TYPE "UDT_WSGConfiguration"
VERSION : 0.1
   STRUCT
      GlobalConfig { ExternalAccessible := 'False'; ExternalVisible := 'False'; ExternalWritable := 'False'} : Struct
         LeftStationExists { ExternalAccessible := 'False'; ExternalVisible := 'False'; ExternalWritable := 'False'} : Bool := TRUE;
         RightStationExists { ExternalAccessible := 'False'; ExternalVisible := 'False'; ExternalWritable := 'False'} : Bool := TRUE;
      END_STRUCT;
      "010" { ExternalAccessible := 'False'; ExternalVisible := 'False'; ExternalWritable := 'False'} : Struct
         Conveyor { ExternalAccessible := 'False'; ExternalVisible := 'False'; ExternalWritable := 'False'; S7_SetPoint := 'False'} : "UDT_ConveyorConfiguration" := (((), ()), (), (), 100, (), 500, 1000, FALSE, ());
         PEC_Eos { ExternalAccessible := 'False'; ExternalVisible := 'False'; ExternalWritable := 'False'; S7_SetPoint := 'False'} : "UDT_PECConfiguration";
         MCO_M01 { ExternalAccessible := 'False'; ExternalVisible := 'False'; ExternalWritable := 'False'; S7_SetPoint := 'False'} : "UDT_AixPlcFullControllerConfiguration";
      END_STRUCT;
      "020" { ExternalAccessible := 'False'; ExternalVisible := 'False'; ExternalWritable := 'False'} : Struct
         Conveyor { ExternalAccessible := 'False'; ExternalVisible := 'False'; ExternalWritable := 'False'; S7_SetPoint := 'False'} : "UDT_ConveyorConfiguration" := (((), ()), (), (), 100, 0, 500, 1000, FALSE, FALSE);
         PEC_EoS { ExternalAccessible := 'False'; ExternalVisible := 'False'; ExternalWritable := 'False'} : "UDT_PECConfiguration";
         MCO_M01 { ExternalAccessible := 'False'; ExternalVisible := 'False'; ExternalWritable := 'False'; S7_SetPoint := 'False'} : "UDT_AixPlcFullControllerConfiguration";
      END_STRUCT;
      "021" { ExternalAccessible := 'False'; ExternalVisible := 'False'; ExternalWritable := 'False'} : Struct
         Conveyor { ExternalAccessible := 'False'; ExternalVisible := 'False'; ExternalWritable := 'False'; S7_SetPoint := 'False'} : "UDT_ConveyorConfiguration" := (((), ()), (), (), 100, 0, 500, 1000, FALSE, FALSE);
         RightAngledTransfer { ExternalAccessible := 'False'; ExternalVisible := 'False'; ExternalWritable := 'False'; S7_SetPoint := 'False'} : "UDT_RATConfiguration";
         MCO_M01 { ExternalAccessible := 'False'; ExternalVisible := 'False'; ExternalWritable := 'False'; S7_SetPoint := 'False'} : "UDT_AixPlcFullControllerConfiguration";
      END_STRUCT;
      "110" { ExternalAccessible := 'False'; ExternalVisible := 'False'; ExternalWritable := 'False'} : Struct
         Conveyor { ExternalAccessible := 'False'; ExternalVisible := 'False'; ExternalWritable := 'False'; S7_SetPoint := 'False'} : "UDT_ConveyorConfiguration" := (((), ()), (), (), (), (), 500, 1000, FALSE, ());
         PEC_Eos { ExternalAccessible := 'False'; ExternalVisible := 'False'; ExternalWritable := 'False'} : "UDT_PECUpdateConfiguration";
         MCO_M01 { ExternalAccessible := 'False'; ExternalVisible := 'False'; ExternalWritable := 'False'} : "UDT_AixPlcFullControllerConfiguration";
      END_STRUCT;
      "120" { ExternalAccessible := 'False'; ExternalVisible := 'False'; ExternalWritable := 'False'} : Struct
         Conveyor { ExternalAccessible := 'False'; ExternalVisible := 'False'; ExternalWritable := 'False'; S7_SetPoint := 'False'} : "UDT_ConveyorConfiguration" := (((), ()), (), (), (), (), 500, 1000, FALSE, ());
         MCO_M01 { ExternalAccessible := 'False'; ExternalVisible := 'False'; ExternalWritable := 'False'} : "UDT_AixPlcFullControllerConfiguration";
      END_STRUCT;
      "130" { ExternalAccessible := 'False'; ExternalVisible := 'False'; ExternalWritable := 'False'} : Struct
         Conveyor { ExternalAccessible := 'False'; ExternalVisible := 'False'; ExternalWritable := 'False'; S7_SetPoint := 'False'} : "UDT_ConveyorConfiguration" := (((), ()), (), (), 100, (), 500, 1000, FALSE, ());
         PEC_Eos { ExternalAccessible := 'False'; ExternalVisible := 'False'; ExternalWritable := 'False'} : "UDT_PECUpdateConfiguration";
         MCO_M01 { ExternalAccessible := 'False'; ExternalVisible := 'False'; ExternalWritable := 'False'} : "UDT_AixPlcFullControllerConfiguration";
      END_STRUCT;
      "140" { ExternalAccessible := 'False'; ExternalVisible := 'False'; ExternalWritable := 'False'} : Struct
         Conveyor { ExternalAccessible := 'False'; ExternalVisible := 'False'; ExternalWritable := 'False'} : "UDT_ConveyorConfiguration" := (((), ()), (), (), 100, 0, 500, 1000, FALSE, FALSE);
         PEC_EoS { ExternalAccessible := 'False'; ExternalVisible := 'False'; ExternalWritable := 'False'} : "UDT_PECConfiguration";
         MCO_M01 { ExternalAccessible := 'False'; ExternalVisible := 'False'; ExternalWritable := 'False'} : "UDT_AixPlcFullControllerConfiguration";
      END_STRUCT;
      "141" { ExternalAccessible := 'False'; ExternalVisible := 'False'; ExternalWritable := 'False'} : Struct
         Conveyor { ExternalAccessible := 'False'; ExternalVisible := 'False'; ExternalWritable := 'False'; S7_SetPoint := 'False'} : "UDT_ConveyorConfiguration" := (((), ()), (), (), 100, 0, 500, 1000, FALSE, FALSE);
         RightAngledTransfer { ExternalAccessible := 'False'; ExternalVisible := 'False'; ExternalWritable := 'False'} : "UDT_RATConfiguration";
         MCO_M01 { ExternalAccessible := 'False'; ExternalVisible := 'False'; ExternalWritable := 'False'} : "UDT_AixPlcFullControllerConfiguration";
      END_STRUCT;
      "150" { ExternalAccessible := 'False'; ExternalVisible := 'False'; ExternalWritable := 'False'} : Struct
         Conveyor { ExternalAccessible := 'False'; ExternalVisible := 'False'; ExternalWritable := 'False'; S7_SetPoint := 'False'} : "UDT_ConveyorConfiguration" := (((), ()), (), (), 100, (), 500, 1000, FALSE, ());
         PEC_Eos { ExternalAccessible := 'False'; ExternalVisible := 'False'; ExternalWritable := 'False'} : "UDT_PECUpdateConfiguration" := (600, 300, 5, 5, (), (), 50, 50, (), (), (), 1, 5, (), (), (), ());
         MCO_M01 { ExternalAccessible := 'False'; ExternalVisible := 'False'; ExternalWritable := 'False'} : "UDT_AixPlcFullControllerConfiguration";
      END_STRUCT;
      "160" { ExternalAccessible := 'False'; ExternalVisible := 'False'; ExternalWritable := 'False'} : Struct
         Conveyor { ExternalAccessible := 'False'; ExternalVisible := 'False'; ExternalWritable := 'False'; S7_SetPoint := 'False'} : "UDT_ConveyorConfiguration" := (((), ()), (), (), 100, 0, 500, 1000, FALSE, FALSE);
         PEC_Eos { ExternalAccessible := 'False'; ExternalVisible := 'False'; ExternalWritable := 'False'} : "UDT_PECUpdateConfiguration" := (600, 300, 5, 5, TRUE, FALSE, 50, 50, 1, 5, 0, 1, 5, FALSE, FALSE, FALSE, FALSE);
         MCO_M01 { ExternalAccessible := 'False'; ExternalVisible := 'False'; ExternalWritable := 'False'} : "UDT_AixPlcFullControllerConfiguration";
      END_STRUCT;
      "170" { ExternalAccessible := 'False'; ExternalVisible := 'False'; ExternalWritable := 'False'} : Struct
         Conveyor { ExternalAccessible := 'False'; ExternalVisible := 'False'; ExternalWritable := 'False'; S7_SetPoint := 'False'} : "UDT_ConveyorConfiguration" := (((), ()), (), (), 100, (), 500, 1000, FALSE, ());
         PEC_Eos { ExternalAccessible := 'False'; ExternalVisible := 'False'; ExternalWritable := 'False'} : "UDT_PECUpdateConfiguration" := (600, 300, 5, 5, (), (), 50, 50, (), (), (), 1, 5, (), (), (), ());
         MCO_M01 { ExternalAccessible := 'False'; ExternalVisible := 'False'; ExternalWritable := 'False'} : "UDT_AixPlcFullControllerConfiguration";
      END_STRUCT;
      "180" { ExternalAccessible := 'False'; ExternalVisible := 'False'; ExternalWritable := 'False'} : Struct
         Conveyor { ExternalAccessible := 'False'; ExternalVisible := 'False'; ExternalWritable := 'False'; S7_SetPoint := 'False'} : "UDT_ConveyorConfiguration" := (((), ()), (), (), 100, (), 500, 1000, FALSE, ());
         PEC_Eos { ExternalAccessible := 'False'; ExternalVisible := 'False'; ExternalWritable := 'False'} : "UDT_PECUpdateConfiguration" := (600, 300, 5, 5, (), (), 50, 50, (), (), (), 1, 5, (), (), (), ());
         MCO_M01 { ExternalAccessible := 'False'; ExternalVisible := 'False'; ExternalWritable := 'False'} : "UDT_AixPlcFullControllerConfiguration";
      END_STRUCT;
      "190" { ExternalAccessible := 'False'; ExternalVisible := 'False'; ExternalWritable := 'False'} : Struct
         Conveyor { ExternalAccessible := 'False'; ExternalVisible := 'False'; ExternalWritable := 'False'; S7_SetPoint := 'False'} : "UDT_ConveyorConfiguration" := (((), ()), (), (), 100, (), 500, 1000, FALSE, ());
         PEC_Eos { ExternalAccessible := 'False'; ExternalVisible := 'False'; ExternalWritable := 'False'} : "UDT_PECUpdateConfiguration" := (600, 300, 5, 5, (), (), 50, 50, (), (), (), 1, 5, (), (), (), ());
         MCO_M01 { ExternalAccessible := 'False'; ExternalVisible := 'False'; ExternalWritable := 'False'} : "UDT_AixPlcFullControllerConfiguration";
      END_STRUCT;
      "210" { ExternalAccessible := 'False'; ExternalVisible := 'False'; ExternalWritable := 'False'} : Struct
         Conveyor { ExternalAccessible := 'False'; ExternalVisible := 'False'; ExternalWritable := 'False'; S7_SetPoint := 'False'} : "UDT_ConveyorConfiguration" := (((), ()), (), (), 100, 0, 500, 1000, FALSE, FALSE);
         PEC_EoS { ExternalAccessible := 'False'; ExternalVisible := 'False'; ExternalWritable := 'False'} : "UDT_PECConfiguration";
         MCO_M01 { ExternalAccessible := 'False'; ExternalVisible := 'False'; ExternalWritable := 'False'} : "UDT_AixPlcFullControllerConfiguration";
      END_STRUCT;
      "211" { ExternalAccessible := 'False'; ExternalVisible := 'False'; ExternalWritable := 'False'} : Struct
         Conveyor { ExternalAccessible := 'False'; ExternalVisible := 'False'; ExternalWritable := 'False'; S7_SetPoint := 'False'} : "UDT_ConveyorConfiguration" := (((), ()), (), (), 100, 0, 500, 1000, FALSE, FALSE);
         RightAngledTransfer { ExternalAccessible := 'False'; ExternalVisible := 'False'; ExternalWritable := 'False'} : "UDT_RATConfiguration";
         MCO_M01 { ExternalAccessible := 'False'; ExternalVisible := 'False'; ExternalWritable := 'False'} : "UDT_AixPlcFullControllerConfiguration";
      END_STRUCT;
      "220" { ExternalAccessible := 'False'; ExternalVisible := 'False'; ExternalWritable := 'False'} : Struct
         Conveyor { ExternalAccessible := 'False'; ExternalVisible := 'False'; ExternalWritable := 'False'} : "UDT_ConveyorConfiguration" := (((), ()), (), (), 100, 0, 500, 1000, FALSE, FALSE);
         PEC_EoS { ExternalAccessible := 'False'; ExternalVisible := 'False'; ExternalWritable := 'False'} : "UDT_PECConfiguration";
         MCO_M01 { ExternalAccessible := 'False'; ExternalVisible := 'False'; ExternalWritable := 'False'} : "UDT_AixPlcFullControllerConfiguration";
      END_STRUCT;
      "221" { ExternalAccessible := 'False'; ExternalVisible := 'False'; ExternalWritable := 'False'} : Struct
         Conveyor { ExternalAccessible := 'False'; ExternalVisible := 'False'; ExternalWritable := 'False'; S7_SetPoint := 'False'} : "UDT_ConveyorConfiguration" := (((), ()), (), (), 100, 0, 500, 1000, FALSE, FALSE);
         RightAngledTransfer { ExternalAccessible := 'False'; ExternalVisible := 'False'; ExternalWritable := 'False'} : "UDT_RATConfiguration";
         MCO_M01 { ExternalAccessible := 'False'; ExternalVisible := 'False'; ExternalWritable := 'False'} : "UDT_AixPlcFullControllerConfiguration";
      END_STRUCT;
      "230" { ExternalAccessible := 'False'; ExternalVisible := 'False'; ExternalWritable := 'False'} : Struct
         Conveyor { ExternalAccessible := 'False'; ExternalVisible := 'False'; ExternalWritable := 'False'; S7_SetPoint := 'False'} : "UDT_ConveyorConfiguration" := (((), ()), (), (), 100, (), 500, 1000, FALSE, ());
         MCO_M01 { ExternalAccessible := 'False'; ExternalVisible := 'False'; ExternalWritable := 'False'} : "UDT_AixPlcFullControllerConfiguration";
      END_STRUCT;
      "310" { ExternalAccessible := 'False'; ExternalVisible := 'False'; ExternalWritable := 'False'} : Struct
         Conveyor { ExternalAccessible := 'False'; ExternalVisible := 'False'; ExternalWritable := 'False'; S7_SetPoint := 'False'} : "UDT_ConveyorConfiguration" := (((), ()), (), (), 100, (), 500, 1000, FALSE, ());
         PEC_Eos { ExternalAccessible := 'False'; ExternalVisible := 'False'; ExternalWritable := 'False'} : "UDT_PECConfiguration" := (600, 300, 5, 5, ());
         MCO_M01 { ExternalAccessible := 'False'; ExternalVisible := 'False'; ExternalWritable := 'False'} : "UDT_AixPlcFullControllerConfiguration";
      END_STRUCT;
      "320" { ExternalAccessible := 'False'; ExternalVisible := 'False'; ExternalWritable := 'False'} : Struct
         Conveyor { ExternalAccessible := 'False'; ExternalVisible := 'False'; ExternalWritable := 'False'; S7_SetPoint := 'False'} : "UDT_ConveyorConfiguration" := (((), ()), (), (), 100, (), 500, 1000, FALSE, ());
         PEC_Eos { ExternalAccessible := 'False'; ExternalVisible := 'False'; ExternalWritable := 'False'} : "UDT_PECConfiguration" := (600, 300, 5, 5, ());
         MCO_M01 { ExternalAccessible := 'False'; ExternalVisible := 'False'; ExternalWritable := 'False'} : "UDT_AixPlcFullControllerConfiguration";
      END_STRUCT;
      "330" { ExternalAccessible := 'False'; ExternalVisible := 'False'; ExternalWritable := 'False'} : Struct
         Conveyor { ExternalAccessible := 'False'; ExternalVisible := 'False'; ExternalWritable := 'False'; S7_SetPoint := 'False'} : "UDT_ConveyorConfiguration" := (((), ()), (), (), 100, (), 500, 1000, FALSE, ());
         PEC_Eos { ExternalAccessible := 'False'; ExternalVisible := 'False'; ExternalWritable := 'False'} : "UDT_PECConfiguration" := (600, 300, 5, 5, ());
         MCO_M01 { ExternalAccessible := 'False'; ExternalVisible := 'False'; ExternalWritable := 'False'} : "UDT_AixPlcFullControllerConfiguration";
      END_STRUCT;
      "340" { ExternalAccessible := 'False'; ExternalVisible := 'False'; ExternalWritable := 'False'} : Struct
         Conveyor { ExternalAccessible := 'False'; ExternalVisible := 'False'; ExternalWritable := 'False'; S7_SetPoint := 'False'} : "UDT_ConveyorConfiguration" := (((), ()), (), (), 100, (), 500, 1000, FALSE, ());
         PEC_Eos { ExternalAccessible := 'False'; ExternalVisible := 'False'; ExternalWritable := 'False'} : "UDT_PECConfiguration" := (600, 300, 5, 5, ());
         MCO_M01 { ExternalAccessible := 'False'; ExternalVisible := 'False'; ExternalWritable := 'False'} : "UDT_AixPlcFullControllerConfiguration";
      END_STRUCT;
      "350" { ExternalAccessible := 'False'; ExternalVisible := 'False'; ExternalWritable := 'False'} : Struct
         Conveyor { ExternalAccessible := 'False'; ExternalVisible := 'False'; ExternalWritable := 'False'; S7_SetPoint := 'False'} : "UDT_ConveyorConfiguration" := (((), ()), (), (), 100, (), 500, 1000, FALSE, ());
         PEC_Eos { ExternalAccessible := 'False'; ExternalVisible := 'False'; ExternalWritable := 'False'} : "UDT_PECConfiguration" := (600, 300, 5, 5, ());
         MCO_M01 { ExternalAccessible := 'False'; ExternalVisible := 'False'; ExternalWritable := 'False'} : "UDT_AixPlcFullControllerConfiguration";
      END_STRUCT;
      "510" { ExternalAccessible := 'False'; ExternalVisible := 'False'; ExternalWritable := 'False'} : Struct
         Conveyor { ExternalAccessible := 'False'; ExternalVisible := 'False'; ExternalWritable := 'False'; S7_SetPoint := 'False'} : "UDT_ConveyorConfiguration" := (((), ()), (), (), 100, (), 500, 1000, FALSE, ());
         MCO_M01 { ExternalAccessible := 'False'; ExternalVisible := 'False'; ExternalWritable := 'False'} : "UDT_AixPlcFullControllerConfiguration";
      END_STRUCT;
      "520" { ExternalAccessible := 'False'; ExternalVisible := 'False'; ExternalWritable := 'False'} : Struct
         Conveyor { ExternalAccessible := 'False'; ExternalVisible := 'False'; ExternalWritable := 'False'; S7_SetPoint := 'False'} : "UDT_ConveyorConfiguration" := (((), ()), (), (), 100, (), 500, 1000, FALSE, ());
         PEC_Eos { ExternalAccessible := 'False'; ExternalVisible := 'False'; ExternalWritable := 'False'; S7_SetPoint := 'False'} : "UDT_PECUpdateConfiguration";
         MCO_M01 { ExternalAccessible := 'False'; ExternalVisible := 'False'; ExternalWritable := 'False'} : "UDT_AixPlcFullControllerConfiguration";
      END_STRUCT;
      "530" { ExternalAccessible := 'False'; ExternalVisible := 'False'; ExternalWritable := 'False'} : Struct
         Conveyor { ExternalAccessible := 'False'; ExternalVisible := 'False'; ExternalWritable := 'False'; S7_SetPoint := 'False'} : "UDT_ConveyorConfiguration" := (((), ()), (), (), 100, (), 500, 1000, FALSE, ());
         PEC_Eos { ExternalAccessible := 'False'; ExternalVisible := 'False'; ExternalWritable := 'False'; S7_SetPoint := 'False'} : "UDT_PECUpdateConfiguration";
         MCO_M01 { ExternalAccessible := 'False'; ExternalVisible := 'False'; ExternalWritable := 'False'} : "UDT_AixPlcFullControllerConfiguration";
      END_STRUCT;
      "540" { ExternalAccessible := 'False'; ExternalVisible := 'False'; ExternalWritable := 'False'} : Struct
         Conveyor { ExternalAccessible := 'False'; ExternalVisible := 'False'; ExternalWritable := 'False'} : "UDT_ConveyorConfiguration" := (((), ()), (), (), 100, 0, 500, 1000, FALSE, FALSE);
         PEC_EoS { ExternalAccessible := 'False'; ExternalVisible := 'False'; ExternalWritable := 'False'} : "UDT_PECConfiguration";
         MCO_M01 { ExternalAccessible := 'False'; ExternalVisible := 'False'; ExternalWritable := 'False'} : "UDT_AixPlcFullControllerConfiguration";
      END_STRUCT;
      "541" { ExternalAccessible := 'False'; ExternalVisible := 'False'; ExternalWritable := 'False'} : Struct
         Conveyor { ExternalAccessible := 'False'; ExternalVisible := 'False'; ExternalWritable := 'False'} : "UDT_ConveyorConfiguration" := (((), ()), (), (), 100, 0, 500, 1000, FALSE, FALSE);
         RightAngledTransfer { ExternalAccessible := 'False'; ExternalVisible := 'False'; ExternalWritable := 'False'} : "UDT_RATConfiguration";
         MCO_M01 { ExternalAccessible := 'False'; ExternalVisible := 'False'; ExternalWritable := 'False'} : "UDT_AixPlcFullControllerConfiguration";
      END_STRUCT;
      "550" { ExternalAccessible := 'False'; ExternalVisible := 'False'; ExternalWritable := 'False'} : Struct
         Conveyor { ExternalAccessible := 'False'; ExternalVisible := 'False'; ExternalWritable := 'False'; S7_SetPoint := 'False'} : "UDT_ConveyorConfiguration" := (((), ()), (), (), 100, (), 500, 1000, FALSE, ());
         PEC_Eos { ExternalAccessible := 'False'; ExternalVisible := 'False'; ExternalWritable := 'False'} : "UDT_PECUpdateConfiguration" := (600, 300, 5, 5, (), (), 50, 50, (), (), (), 1, 5, (), (), (), ());
         MCO_M01 { ExternalAccessible := 'False'; ExternalVisible := 'False'; ExternalWritable := 'False'} : "UDT_AixPlcFullControllerConfiguration";
      END_STRUCT;
      "560" { ExternalAccessible := 'False'; ExternalVisible := 'False'; ExternalWritable := 'False'} : Struct
         Conveyor { ExternalAccessible := 'False'; ExternalVisible := 'False'; ExternalWritable := 'False'; S7_SetPoint := 'False'} : "UDT_ConveyorConfiguration" := (((), ()), (), (), 100, 0, 500, 1000, FALSE, FALSE);
         PEC_Eos { ExternalAccessible := 'False'; ExternalVisible := 'False'; ExternalWritable := 'False'} : "UDT_PECUpdateConfiguration" := (600, 300, 5, 5, TRUE, FALSE, 50, 50, 1, 5, 0, 1, 5, FALSE, FALSE, FALSE, FALSE);
         MCO_M01 { ExternalAccessible := 'False'; ExternalVisible := 'False'; ExternalWritable := 'False'} : "UDT_AixPlcFullControllerConfiguration";
      END_STRUCT;
      "570" { ExternalAccessible := 'False'; ExternalVisible := 'False'; ExternalWritable := 'False'} : Struct
         Conveyor { ExternalAccessible := 'False'; ExternalVisible := 'False'; ExternalWritable := 'False'; S7_SetPoint := 'False'} : "UDT_ConveyorConfiguration" := (((), ()), (), (), 100, (), 500, 1000, FALSE, ());
         PEC_Eos { ExternalAccessible := 'False'; ExternalVisible := 'False'; ExternalWritable := 'False'} : "UDT_PECUpdateConfiguration" := (600, 300, 5, 5, (), (), 50, 50, (), (), (), 1, 5, (), (), (), ());
         MCO_M01 { ExternalAccessible := 'False'; ExternalVisible := 'False'; ExternalWritable := 'False'} : "UDT_AixPlcFullControllerConfiguration";
      END_STRUCT;
      "580" { ExternalAccessible := 'False'; ExternalVisible := 'False'; ExternalWritable := 'False'} : Struct
         Conveyor { ExternalAccessible := 'False'; ExternalVisible := 'False'; ExternalWritable := 'False'; S7_SetPoint := 'False'} : "UDT_ConveyorConfiguration" := (((), ()), (), (), 100, (), 500, 1000, FALSE, ());
         PEC_Eos { ExternalAccessible := 'False'; ExternalVisible := 'False'; ExternalWritable := 'False'} : "UDT_PECUpdateConfiguration" := (600, 300, 5, 5, (), (), 50, 50, (), (), (), 1, 5, (), (), (), ());
         MCO_M01 { ExternalAccessible := 'False'; ExternalVisible := 'False'; ExternalWritable := 'False'} : "UDT_AixPlcFullControllerConfiguration";
      END_STRUCT;
      "590" { ExternalAccessible := 'False'; ExternalVisible := 'False'; ExternalWritable := 'False'} : Struct
         Conveyor { ExternalAccessible := 'False'; ExternalVisible := 'False'; ExternalWritable := 'False'; S7_SetPoint := 'False'} : "UDT_ConveyorConfiguration" := (((), ()), (), (), 100, (), 500, 1000, FALSE, ());
         PEC_Eos { ExternalAccessible := 'False'; ExternalVisible := 'False'; ExternalWritable := 'False'} : "UDT_PECUpdateConfiguration" := (600, 300, 5, 5, (), (), 50, 50, (), (), (), 1, 5, (), (), (), ());
         MCO_M01 { ExternalAccessible := 'False'; ExternalVisible := 'False'; ExternalWritable := 'False'} : "UDT_AixPlcFullControllerConfiguration";
      END_STRUCT;
      "610" { ExternalAccessible := 'False'; ExternalVisible := 'False'; ExternalWritable := 'False'} : Struct
         Conveyor { ExternalAccessible := 'False'; ExternalVisible := 'False'; ExternalWritable := 'False'; S7_SetPoint := 'False'} : "UDT_ConveyorConfiguration" := (((), ()), (), (), 100, 0, 500, 1000, FALSE, FALSE);
         PEC_EoS { ExternalAccessible := 'False'; ExternalVisible := 'False'; ExternalWritable := 'False'} : "UDT_PECConfiguration";
         MCO_M01 { ExternalAccessible := 'False'; ExternalVisible := 'False'; ExternalWritable := 'False'} : "UDT_AixPlcFullControllerConfiguration";
      END_STRUCT;
      "611" { ExternalAccessible := 'False'; ExternalVisible := 'False'; ExternalWritable := 'False'} : Struct
         Conveyor { ExternalAccessible := 'False'; ExternalVisible := 'False'; ExternalWritable := 'False'; S7_SetPoint := 'False'} : "UDT_ConveyorConfiguration" := (((), ()), (), (), 100, 0, 500, 1000, FALSE, FALSE);
         RightAngledTransfer { ExternalAccessible := 'False'; ExternalVisible := 'False'; ExternalWritable := 'False'} : "UDT_RATConfiguration";
         MCO_M01 { ExternalAccessible := 'False'; ExternalVisible := 'False'; ExternalWritable := 'False'} : "UDT_AixPlcFullControllerConfiguration";
      END_STRUCT;
      "620" { ExternalAccessible := 'False'; ExternalVisible := 'False'; ExternalWritable := 'False'} : Struct
         Conveyor { ExternalAccessible := 'False'; ExternalVisible := 'False'; ExternalWritable := 'False'} : "UDT_ConveyorConfiguration" := (((), ()), (), (), 100, 0, 500, 1000, FALSE, FALSE);
         PEC_EoS { ExternalAccessible := 'False'; ExternalVisible := 'False'; ExternalWritable := 'False'} : "UDT_PECConfiguration";
         MCO_M01 { ExternalAccessible := 'False'; ExternalVisible := 'False'; ExternalWritable := 'False'} : "UDT_AixPlcFullControllerConfiguration";
      END_STRUCT;
      "621" { ExternalAccessible := 'False'; ExternalVisible := 'False'; ExternalWritable := 'False'} : Struct
         Conveyor { ExternalAccessible := 'False'; ExternalVisible := 'False'; ExternalWritable := 'False'; S7_SetPoint := 'False'} : "UDT_ConveyorConfiguration" := (((), ()), (), (), 100, 0, 500, 1000, FALSE, FALSE);
         RightAngledTransfer { ExternalAccessible := 'False'; ExternalVisible := 'False'; ExternalWritable := 'False'} : "UDT_RATConfiguration";
         MCO_M01 { ExternalAccessible := 'False'; ExternalVisible := 'False'; ExternalWritable := 'False'} : "UDT_AixPlcFullControllerConfiguration";
      END_STRUCT;
      "630" { ExternalAccessible := 'False'; ExternalVisible := 'False'; ExternalWritable := 'False'} : Struct
         Conveyor { ExternalAccessible := 'False'; ExternalVisible := 'False'; ExternalWritable := 'False'; S7_SetPoint := 'False'} : "UDT_ConveyorConfiguration" := (((), ()), (), (), 100, (), 500, 1000, FALSE, ());
         MCO_M01 { ExternalAccessible := 'False'; ExternalVisible := 'False'; ExternalWritable := 'False'} : "UDT_AixPlcFullControllerConfiguration";
      END_STRUCT;
      "710" { ExternalAccessible := 'False'; ExternalVisible := 'False'; ExternalWritable := 'False'} : Struct
         Conveyor { ExternalAccessible := 'False'; ExternalVisible := 'False'; ExternalWritable := 'False'; S7_SetPoint := 'False'} : "UDT_ConveyorConfiguration" := (((), ()), (), (), 100, (), 500, 1000, FALSE, ());
         PEC_Eos { ExternalAccessible := 'False'; ExternalVisible := 'False'; ExternalWritable := 'False'} : "UDT_PECConfiguration" := (600, 300, 5, 5, ());
         MCO_M01 { ExternalAccessible := 'False'; ExternalVisible := 'False'; ExternalWritable := 'False'} : "UDT_AixPlcFullControllerConfiguration";
      END_STRUCT;
      "720" { ExternalAccessible := 'False'; ExternalVisible := 'False'; ExternalWritable := 'False'} : Struct
         Conveyor { ExternalAccessible := 'False'; ExternalVisible := 'False'; ExternalWritable := 'False'; S7_SetPoint := 'False'} : "UDT_ConveyorConfiguration" := (((), ()), (), (), 100, (), 500, 1000, FALSE, ());
         PEC_Eos { ExternalAccessible := 'False'; ExternalVisible := 'False'; ExternalWritable := 'False'} : "UDT_PECConfiguration" := (600, 300, 5, 5, ());
         MCO_M01 { ExternalAccessible := 'False'; ExternalVisible := 'False'; ExternalWritable := 'False'} : "UDT_AixPlcFullControllerConfiguration";
      END_STRUCT;
      "730" { ExternalAccessible := 'False'; ExternalVisible := 'False'; ExternalWritable := 'False'} : Struct
         Conveyor { ExternalAccessible := 'False'; ExternalVisible := 'False'; ExternalWritable := 'False'; S7_SetPoint := 'False'} : "UDT_ConveyorConfiguration" := (((), ()), (), (), 100, (), 500, 1000, FALSE, ());
         PEC_Eos { ExternalAccessible := 'False'; ExternalVisible := 'False'; ExternalWritable := 'False'} : "UDT_PECConfiguration" := (600, 300, 5, 5, ());
         MCO_M01 { ExternalAccessible := 'False'; ExternalVisible := 'False'; ExternalWritable := 'False'} : "UDT_AixPlcFullControllerConfiguration";
      END_STRUCT;
      "740" { ExternalAccessible := 'False'; ExternalVisible := 'False'; ExternalWritable := 'False'} : Struct
         Conveyor { ExternalAccessible := 'False'; ExternalVisible := 'False'; ExternalWritable := 'False'; S7_SetPoint := 'False'} : "UDT_ConveyorConfiguration" := (((), ()), (), (), 100, (), 500, 1000, FALSE, ());
         PEC_Eos { ExternalAccessible := 'False'; ExternalVisible := 'False'; ExternalWritable := 'False'} : "UDT_PECConfiguration" := (600, 300, 5, 5, ());
         MCO_M01 { ExternalAccessible := 'False'; ExternalVisible := 'False'; ExternalWritable := 'False'} : "UDT_AixPlcFullControllerConfiguration";
      END_STRUCT;
      "750" { ExternalAccessible := 'False'; ExternalVisible := 'False'; ExternalWritable := 'False'} : Struct
         Conveyor { ExternalAccessible := 'False'; ExternalVisible := 'False'; ExternalWritable := 'False'; S7_SetPoint := 'False'} : "UDT_ConveyorConfiguration" := (((), ()), (), (), 100, (), 500, 1000, FALSE, ());
         PEC_Eos { ExternalAccessible := 'False'; ExternalVisible := 'False'; ExternalWritable := 'False'} : "UDT_PECConfiguration" := (600, 300, 5, 5, ());
         MCO_M01 { ExternalAccessible := 'False'; ExternalVisible := 'False'; ExternalWritable := 'False'} : "UDT_AixPlcFullControllerConfiguration";
      END_STRUCT;
   END_STRUCT;

END_TYPE

TYPE "UDT_NerakLiftPO"
VERSION : 0.1
   STRUCT
      qx_PowerRelease { ExternalAccessible := 'False'; ExternalVisible := 'False'; ExternalWritable := 'False'} : Bool;   // Release main contactor 17Q1
      "qx_spare_0.1" { ExternalAccessible := 'False'; ExternalVisible := 'False'; ExternalWritable := 'False'} : Bool;
      qx_ReadyLamp { ExternalAccessible := 'False'; ExternalVisible := 'False'; ExternalWritable := 'False'} : Bool;   // LED lamp GREEN - Ready
      "qx_spare_0.3" { ExternalAccessible := 'False'; ExternalVisible := 'False'; ExternalWritable := 'False'} : Bool;
      qx_FaultLamp { ExternalAccessible := 'False'; ExternalVisible := 'False'; ExternalWritable := 'False'} : Bool;   // LED lamp RED - Fault
      "qx_spare_0.5" { ExternalAccessible := 'False'; ExternalVisible := 'False'; ExternalWritable := 'False'} : Bool;
      "qx_spare_0.6" { ExternalAccessible := 'False'; ExternalVisible := 'False'; ExternalWritable := 'False'} : Bool;
      "qx_spare_0.7" { ExternalAccessible := 'False'; ExternalVisible := 'False'; ExternalWritable := 'False'} : Bool;
   END_STRUCT;

END_TYPE

TYPE "UDT_NerakLiftPI"
VERSION : 0.1
   STRUCT
      ix_PowerOK { ExternalAccessible := 'False'; ExternalVisible := 'False'; ExternalWritable := 'False'} : Bool;   // -10F1, -12F1 and -12Q1 are switched ON
      ix_ManualDown { ExternalAccessible := 'False'; ExternalVisible := 'False'; ExternalWritable := 'False'} : Bool;   // Push button manual DOWN
      ix_ManualMode { ExternalAccessible := 'False'; ExternalVisible := 'False'; ExternalWritable := 'False'} : Bool;   // Key switch manual mode
      ix_FaultReset { ExternalAccessible := 'False'; ExternalVisible := 'False'; ExternalWritable := 'False'} : Bool;   // Push button reset fault
      ix_AutomaticMode { ExternalAccessible := 'False'; ExternalVisible := 'False'; ExternalWritable := 'False'} : Bool;   // Key switch automatic mode
      "ix_spare_0.5" { ExternalAccessible := 'False'; ExternalVisible := 'False'; ExternalWritable := 'False'} : Bool;
      ix_ManualUp { ExternalAccessible := 'False'; ExternalVisible := 'False'; ExternalWritable := 'False'} : Bool;   // Push button manual UP
      ix_B11ColisionControl { ExternalAccessible := 'False'; ExternalVisible := 'False'; ExternalWritable := 'False'} : Bool;   // Sensor -B11 Collisiion control top
      ix_B1Infeed { ExternalAccessible := 'False'; ExternalVisible := 'False'; ExternalWritable := 'False'} : Bool;   // Sensor  -B1 Infeed occupied
      "ix_B3.3FallingThrought" { ExternalAccessible := 'False'; ExternalVisible := 'False'; ExternalWritable := 'False'} : Bool;   // Sensor -B3.3 Falling through control
      ix_B2_CollisionControl { ExternalAccessible := 'False'; ExternalVisible := 'False'; ExternalWritable := 'False'} : Bool;   // Sensor -B2 Collision at infeed
      ix_B4TailbackControlFront { ExternalAccessible := 'False'; ExternalVisible := 'False'; ExternalWritable := 'False'} : Bool;   // Sensor -B4 Outfeed occupied
      "ix_B3.1FallingThrought" { ExternalAccessible := 'False'; ExternalVisible := 'False'; ExternalWritable := 'False'} : Bool;   // Sensor -B3.1 Falling through control
      ix_B5TailbackControlBack { ExternalAccessible := 'False'; ExternalVisible := 'False'; ExternalWritable := 'False'} : Bool;   // Sensor -B4 Product before Outfeed
      "ix_B3.2FallingThrought" { ExternalAccessible := 'False'; ExternalVisible := 'False'; ExternalWritable := 'False'} : Bool;   // Sensor -B3.2 Falling through control
      ix_B10_PlatforninPosition { ExternalAccessible := 'False'; ExternalVisible := 'False'; ExternalWritable := 'False'} : Bool;   // Sensor -B10 Platform in position to start infeed
      ix_DoorSwitchBottom { ExternalAccessible := 'False'; ExternalVisible := 'False'; ExternalWritable := 'False'} : Bool;   // Door switch bottom -16S3 diagnostic
      "ix_spare_2.1" { ExternalAccessible := 'False'; ExternalVisible := 'False'; ExternalWritable := 'False'} : Bool;
      ix_DoorSwitchTop { ExternalAccessible := 'False'; ExternalVisible := 'False'; ExternalWritable := 'False'} : Bool;   // Door switch up -16S4 diagnostic
      "ix_spare_2.3" { ExternalAccessible := 'False'; ExternalVisible := 'False'; ExternalWritable := 'False'} : Bool;
      "ix_spare_2.4" { ExternalAccessible := 'False'; ExternalVisible := 'False'; ExternalWritable := 'False'} : Bool;
      "ix_spare_2.5" { ExternalAccessible := 'False'; ExternalVisible := 'False'; ExternalWritable := 'False'} : Bool;
      "ix_spare_2.6" { ExternalAccessible := 'False'; ExternalVisible := 'False'; ExternalWritable := 'False'} : Bool;
      "ix_spare_2.7" { ExternalAccessible := 'False'; ExternalVisible := 'False'; ExternalWritable := 'False'} : Bool;
   END_STRUCT;

END_TYPE

TYPE "UDT_NerakLiftConfiguration"
VERSION : 0.1
   STRUCT
      Mode { ExternalAccessible := 'False'; ExternalVisible := 'False'; ExternalWritable := 'False'} : Int;   // 1 - lowering mode 2 - lifting mode
      CollisionSensorDelayOn { ExternalAccessible := 'False'; ExternalVisible := 'False'; ExternalWritable := 'False'} : UDInt;   // Collision sensor delay on
      CollisionSensorDelayOff { ExternalAccessible := 'False'; ExternalVisible := 'False'; ExternalWritable := 'False'} : UDInt;   // Collision sensor delay off
      FallingThroughSensorDelayOn { ExternalAccessible := 'False'; ExternalVisible := 'False'; ExternalWritable := 'False'} : UDInt;   // Falling through sensor delay on
      FallingThroughSensorDelayOff { ExternalAccessible := 'False'; ExternalVisible := 'False'; ExternalWritable := 'False'} : UDInt;   // Falling through sensor delay off
      TailbackControlFrontSensorDelayOn { ExternalAccessible := 'False'; ExternalVisible := 'False'; ExternalWritable := 'False'} : UDInt;   // Tailback control front sensor delay on
      TailbackControlFrontSensorDelayOff { ExternalAccessible := 'False'; ExternalVisible := 'False'; ExternalWritable := 'False'} : UDInt;   // Tailback control front sensor delay off
      TailbackControlRearSensorDelayOn { ExternalAccessible := 'False'; ExternalVisible := 'False'; ExternalWritable := 'False'} : UDInt;   // Tailback control rear sensor delay on
      TailbackControlRearSensorDelayOff { ExternalAccessible := 'False'; ExternalVisible := 'False'; ExternalWritable := 'False'} : UDInt;   // Tailback control rear sensor delay off
      PlatformPositionSensorDelayOn { ExternalAccessible := 'False'; ExternalVisible := 'False'; ExternalWritable := 'False'} : UDInt;   // Platform position sensor delay on
      PlatformPositionSensorDelayOff { ExternalAccessible := 'False'; ExternalVisible := 'False'; ExternalWritable := 'False'} : UDInt;   // Platform position sensor delay off
      PlatformLength { ExternalAccessible := 'False'; ExternalVisible := 'False'; ExternalWritable := 'False'} : Int := 759;   // Platform length [mm]
      Length { ExternalAccessible := 'False'; ExternalVisible := 'False'; ExternalWritable := 'False'} : DInt := 6000;   // Distance to be traveled by the package from start to end[mm]
      EnergySaveLength { ExternalAccessible := 'False'; ExternalVisible := 'False'; ExternalWritable := 'False'} : DInt := 10000;   // Distance to run before energy saving is activated [cm]
      PEC_EoSDistanceOffset { ExternalAccessible := 'False'; ExternalVisible := 'False'; ExternalWritable := 'False'} : DInt := 300;   // Position to stop during dieback [mm]
      CascadeTimeOnDelay { ExternalAccessible := 'False'; ExternalVisible := 'False'; ExternalWritable := 'False'} : UDInt := 200;   // Cascade start delay
      FirstConveyorToStart { ExternalAccessible := 'False'; ExternalVisible := 'False'; ExternalWritable := 'False'} : Bool := FALSE;   // Lift first to start in cascade
      SpeedSetpointNominal { ExternalAccessible := 'False'; ExternalVisible := 'False'; ExternalWritable := 'False'} : Int := 1000;   // Speed setpoint nominal
      Energy { ExternalAccessible := 'False'; ExternalVisible := 'False'; ExternalWritable := 'False'} : Bool := TRUE;   // TRUE when energy saving mode enable
   END_STRUCT;

END_TYPE

TYPE "UDT_WSGCommunicationWES"
VERSION : 0.1
   STRUCT
      LeftWorkstation : Struct   // Communication with left side of station
         StartIndexing : Bool;   // Request to start indexing
         Station1 : Struct
            Gin : Int;   // Message from station1
            Barcode : String;
            Error : Bool;
            ReadyForPush : Bool;   // Request to start automatic push out
         END_STRUCT;
         Station2 : Struct
            Gin : Int;   // Message from station1
            Barcode : String;
            Error : Bool;
            ReadyForPush : Bool;   // Request to start automatic push out
         END_STRUCT;
         Station3 : Struct
            Gin : Int;   // Message from station1
            Barcode : String;
            Error : Bool;
            ReadyForPush : Bool;   // Request to start automatic push out
         END_STRUCT;
         Station4 : Struct
            Gin : Int;   // Message from station1
            Barcode : String;
            Error : Bool;
            ReadyForPush : Bool;   // Request to start automatic push out
         END_STRUCT;
         Station5 : Struct
            Gin : Int;   // Message from station1
            Barcode : String;
            Error : Bool;
            ReadyForPush : Bool;   // Request to start automatic push out
         END_STRUCT;
      END_STRUCT;
      RightWorkstation : Struct   // Communication with left side of station
         StartIndexing : Bool;   // Request to start indexing
         Station1 : Struct
            Gin : Int;   // Message from station1
            Barcode : String;
            Error : Bool;
            ReadyForPush : Bool;   // Request to start automatic push out
         END_STRUCT;
         Station2 : Struct
            Gin : Int;   // Message from station1
            Barcode : String;
            Error : Bool;
            ReadyForPush : Bool;   // Request to start automatic push out
         END_STRUCT;
         Station3 : Struct
            Gin : Int;   // Message from station1
            Barcode : String;
            Error : Bool;
            ReadyForPush : Bool;   // Request to start automatic push out
         END_STRUCT;
         Station4 : Struct
            Gin : Int;   // Message from station1
            Barcode : String;
            Error : Bool;
            ReadyForPush : Bool;   // Request to start automatic push out
         END_STRUCT;
         Station5 : Struct
            Gin : Int;   // Message from station1
            Barcode : String;
            Error : Bool;
            ReadyForPush : Bool;   // Request to start automatic push out
         END_STRUCT;
      END_STRUCT;
   END_STRUCT;

END_TYPE

TYPE "UDT_WSGCommonStatus"
VERSION : 0.1
   STRUCT
      "010" { S7_SetPoint := 'False'} : "UDT_CommonStatus";
      "020" : "UDT_CommonStatus";
      "021" : "UDT_CommonStatus";
      "110" { S7_SetPoint := 'False'} : "UDT_CommonStatus";
      "120" { S7_SetPoint := 'False'} : "UDT_CommonStatus";
      "130" { S7_SetPoint := 'False'} : "UDT_CommonStatus";
      "140" : "UDT_CommonStatus";
      "141" : "UDT_CommonStatus";
      "150" : "UDT_CommonStatus";
      "160" : "UDT_CommonStatus";
      "170" : "UDT_CommonStatus";
      "180" : "UDT_CommonStatus";
      "190" : "UDT_CommonStatus";
      "210" : "UDT_CommonStatus";
      "211" : "UDT_CommonStatus";
      "220" : "UDT_CommonStatus";
      "221" : "UDT_CommonStatus";
      "230" { S7_SetPoint := 'False'} : "UDT_CommonStatus";
      "310" : "UDT_CommonStatus";
      "320" : "UDT_CommonStatus";
      "330" : "UDT_CommonStatus";
      "340" : "UDT_CommonStatus";
      "350" : "UDT_CommonStatus";
      "510" { S7_SetPoint := 'False'} : "UDT_CommonStatus";
      "520" { S7_SetPoint := 'False'} : "UDT_CommonStatus";
      "530" { S7_SetPoint := 'False'} : "UDT_CommonStatus";
      "540" : "UDT_CommonStatus";
      "541" : "UDT_CommonStatus";
      "550" : "UDT_CommonStatus";
      "560" : "UDT_CommonStatus";
      "570" : "UDT_CommonStatus";
      "580" : "UDT_CommonStatus";
      "590" : "UDT_CommonStatus";
      "610" : "UDT_CommonStatus";
      "611" : "UDT_CommonStatus";
      "620" : "UDT_CommonStatus";
      "621" : "UDT_CommonStatus";
      "630" { S7_SetPoint := 'False'} : "UDT_CommonStatus";
      "710" : "UDT_CommonStatus";
      "720" : "UDT_CommonStatus";
      "730" : "UDT_CommonStatus";
      "740" : "UDT_CommonStatus";
      "750" : "UDT_CommonStatus";
   END_STRUCT;

END_TYPE

TYPE "UDT_WSGStatus"
VERSION : 0.1
   STRUCT
      "010" : Struct
         Conveyor { S7_SetPoint := 'False'} : "UDT_ConveyorStatus";
         PEC_EoS : "UDT_PECStatus";
         MCO_M01 : "UDT_AixControllerStatus";
      END_STRUCT;
      "020" : Struct
         Conveyor { S7_SetPoint := 'False'} : "UDT_ConveyorStatus";
         PEC_EoS : "UDT_PECStatus";
         MCO_M01 { S7_SetPoint := 'False'} : "UDT_AixControllerStatus";
      END_STRUCT;
      "021" : Struct
         RightAngledTransfer { S7_SetPoint := 'False'} : "UDT_RATStatus";
         MCO_M01 { S7_SetPoint := 'False'} : "UDT_AixControllerStatus";
      END_STRUCT;
      "110" : Struct
         Conveyor { S7_SetPoint := 'False'} : "UDT_ConveyorStatus";
         PEC_EoS : "UDT_PECUpdateStatus";
         MCO_M01 { S7_SetPoint := 'False'} : "UDT_AixControllerStatus";
      END_STRUCT;
      "120" : Struct
         Conveyor { S7_SetPoint := 'False'} : "UDT_ConveyorStatus";
         PEC_EoS : "UDT_PECStatus";
         MCO_M01 { S7_SetPoint := 'False'} : "UDT_AixControllerStatus";
      END_STRUCT;
      "130" : Struct
         Conveyor { S7_SetPoint := 'False'} : "UDT_ConveyorStatus";
         PEC_EoS : "UDT_PECUpdateStatus";
         MCO_M01 { S7_SetPoint := 'False'} : "UDT_AixControllerStatus";
      END_STRUCT;
      "140" : Struct
         Conveyor { S7_SetPoint := 'False'} : "UDT_ConveyorStatus";
         PEC_EoS : "UDT_PECStatus";
         MCO_M01 { S7_SetPoint := 'False'} : "UDT_AixControllerStatus";
      END_STRUCT;
      "141" : Struct
         RightAngledTransfer { S7_SetPoint := 'False'} : "UDT_RATStatus";
         MCO_M01 { S7_SetPoint := 'False'} : "UDT_AixControllerStatus";
      END_STRUCT;
      "150" : Struct
         Conveyor { S7_SetPoint := 'False'} : "UDT_ConveyorStatus";
         PEC_EoS : "UDT_PECUpdateStatus";
         MCO_M01 { S7_SetPoint := 'False'} : "UDT_AixControllerStatus";
      END_STRUCT;
      "160" : Struct
         Conveyor { S7_SetPoint := 'False'} : "UDT_ConveyorStatus";
         PEC_EoS : "UDT_PECUpdateStatus";
         MCO_M01 { S7_SetPoint := 'False'} : "UDT_AixControllerStatus";
      END_STRUCT;
      "170" : Struct
         Conveyor { S7_SetPoint := 'False'} : "UDT_ConveyorStatus";
         PEC_EoS : "UDT_PECUpdateStatus";
         MCO_M01 { S7_SetPoint := 'False'} : "UDT_AixControllerStatus";
      END_STRUCT;
      "180" : Struct
         Conveyor { S7_SetPoint := 'False'} : "UDT_ConveyorStatus";
         PEC_EoS : "UDT_PECUpdateStatus";
         MCO_M01 { S7_SetPoint := 'False'} : "UDT_AixControllerStatus";
      END_STRUCT;
      "190" : Struct
         Conveyor { S7_SetPoint := 'False'} : "UDT_ConveyorStatus";
         PEC_EoS : "UDT_PECUpdateStatus";
         MCO_M01 { S7_SetPoint := 'False'} : "UDT_AixControllerStatus";
      END_STRUCT;
      "210" : Struct
         Conveyor { S7_SetPoint := 'False'} : "UDT_ConveyorStatus";
         PEC_EoS { S7_SetPoint := 'False'} : "UDT_PECStatus";
         MCO_M01 { S7_SetPoint := 'False'} : "UDT_AixControllerStatus";
      END_STRUCT;
      "211" : Struct
         RightAngledTransfer { S7_SetPoint := 'False'} : "UDT_RATStatus";
         MCO_M01 { S7_SetPoint := 'False'} : "UDT_AixControllerStatus";
      END_STRUCT;
      "220" : Struct
         Conveyor { S7_SetPoint := 'False'} : "UDT_ConveyorStatus";
         PEC_EoS { S7_SetPoint := 'False'} : "UDT_PECStatus";
         MCO_M01 { S7_SetPoint := 'False'} : "UDT_AixControllerStatus";
      END_STRUCT;
      "221" : Struct
         RightAngledTransfer { S7_SetPoint := 'False'} : "UDT_RATStatus";
         MCO_M01 { S7_SetPoint := 'False'} : "UDT_AixControllerStatus";
      END_STRUCT;
      "230" : Struct
         Conveyor { S7_SetPoint := 'False'} : "UDT_ConveyorStatus";
         MCO_M01 { S7_SetPoint := 'False'} : "UDT_AixControllerStatus";
      END_STRUCT;
      "310" : Struct
         Conveyor { S7_SetPoint := 'False'} : "UDT_ConveyorStatus";
         PEC_EoS : "UDT_PECStatus";
         MCO_M01 { S7_SetPoint := 'False'} : "UDT_AixControllerStatus";
      END_STRUCT;
      "320" : Struct
         Conveyor { S7_SetPoint := 'False'} : "UDT_ConveyorStatus";
         PEC_EoS : "UDT_PECStatus";
         MCO_M01 { S7_SetPoint := 'False'} : "UDT_AixControllerStatus";
      END_STRUCT;
      "330" : Struct
         Conveyor { S7_SetPoint := 'False'} : "UDT_ConveyorStatus";
         PEC_EoS : "UDT_PECStatus";
         MCO_M01 { S7_SetPoint := 'False'} : "UDT_AixControllerStatus";
      END_STRUCT;
      "340" : Struct
         Conveyor { S7_SetPoint := 'False'} : "UDT_ConveyorStatus";
         PEC_EoS { S7_SetPoint := 'False'} : "UDT_PECStatus";
         MCO_M01 { S7_SetPoint := 'False'} : "UDT_AixControllerStatus";
      END_STRUCT;
      "350" : Struct
         Conveyor { S7_SetPoint := 'False'} : "UDT_ConveyorStatus";
         PEC_EoS : "UDT_PECStatus";
         MCO_M01 { S7_SetPoint := 'False'} : "UDT_AixControllerStatus";
      END_STRUCT;
      "510" : Struct
         Conveyor { S7_SetPoint := 'False'} : "UDT_ConveyorStatus";
         MCO_M01 { S7_SetPoint := 'False'} : "UDT_AixControllerStatus";
      END_STRUCT;
      "520" : Struct
         Conveyor { S7_SetPoint := 'False'} : "UDT_ConveyorStatus";
         PEC_EoS : "UDT_PECUpdateStatus";
         MCO_M01 { S7_SetPoint := 'False'} : "UDT_AixControllerStatus";
      END_STRUCT;
      "530" : Struct
         Conveyor { S7_SetPoint := 'False'} : "UDT_ConveyorStatus";
         PEC_EoS : "UDT_PECUpdateStatus";
         MCO_M01 { S7_SetPoint := 'False'} : "UDT_AixControllerStatus";
      END_STRUCT;
      "540" : Struct
         Conveyor { S7_SetPoint := 'False'} : "UDT_ConveyorStatus";
         PEC_EoS : "UDT_PECStatus";
         MCO_M01 { S7_SetPoint := 'False'} : "UDT_AixControllerStatus";
      END_STRUCT;
      "541" : Struct
         RightAngledTransfer { S7_SetPoint := 'False'} : "UDT_RATStatus";
         MCO_M01 { S7_SetPoint := 'False'} : "UDT_AixControllerStatus";
      END_STRUCT;
      "550" : Struct
         Conveyor { S7_SetPoint := 'False'} : "UDT_ConveyorStatus";
         PEC_EoS : "UDT_PECUpdateStatus";
         MCO_M01 { S7_SetPoint := 'False'} : "UDT_AixControllerStatus";
      END_STRUCT;
      "560" : Struct
         Conveyor { S7_SetPoint := 'False'} : "UDT_ConveyorStatus";
         PEC_EoS : "UDT_PECUpdateStatus";
         MCO_M01 : "UDT_AixControllerStatus";
      END_STRUCT;
      "570" : Struct
         Conveyor { S7_SetPoint := 'False'} : "UDT_ConveyorStatus";
         PEC_EoS : "UDT_PECUpdateStatus";
         MCO_M01 { S7_SetPoint := 'False'} : "UDT_AixControllerStatus";
      END_STRUCT;
      "580" : Struct
         Conveyor { S7_SetPoint := 'False'} : "UDT_ConveyorStatus";
         PEC_EoS : "UDT_PECUpdateStatus";
         MCO_M01 { S7_SetPoint := 'False'} : "UDT_AixControllerStatus";
      END_STRUCT;
      "590" : Struct
         Conveyor { S7_SetPoint := 'False'} : "UDT_ConveyorStatus";
         PEC_EoS : "UDT_PECUpdateStatus";
         MCO_M01 { S7_SetPoint := 'False'} : "UDT_AixControllerStatus";
      END_STRUCT;
      "610" : Struct
         Conveyor { S7_SetPoint := 'False'} : "UDT_ConveyorStatus";
         PEC_EoS { S7_SetPoint := 'False'} : "UDT_PECStatus";
         MCO_M01 { S7_SetPoint := 'False'} : "UDT_AixControllerStatus";
      END_STRUCT;
      "611" : Struct
         RightAngledTransfer { S7_SetPoint := 'False'} : "UDT_RATStatus";
         MCO_M01 { S7_SetPoint := 'False'} : "UDT_AixControllerStatus";
      END_STRUCT;
      "620" : Struct
         Conveyor { S7_SetPoint := 'False'} : "UDT_ConveyorStatus";
         PEC_EoS { S7_SetPoint := 'False'} : "UDT_PECStatus";
         MCO_M01 { S7_SetPoint := 'False'} : "UDT_AixControllerStatus";
      END_STRUCT;
      "621" : Struct
         RightAngledTransfer { S7_SetPoint := 'False'} : "UDT_RATStatus";
         MCO_M01 : "UDT_AixControllerStatus";
      END_STRUCT;
      "630" : Struct
         Conveyor { S7_SetPoint := 'False'} : "UDT_ConveyorStatus";
         MCO_M01 { S7_SetPoint := 'False'} : "UDT_AixControllerStatus";
      END_STRUCT;
      "710" : Struct
         Conveyor { S7_SetPoint := 'False'} : "UDT_ConveyorStatus";
         PEC_EoS : "UDT_PECStatus";
         MCO_M01 { S7_SetPoint := 'False'} : "UDT_AixControllerStatus";
      END_STRUCT;
      "720" : Struct
         Conveyor { S7_SetPoint := 'False'} : "UDT_ConveyorStatus";
         PEC_EoS : "UDT_PECStatus";
         MCO_M01 : "UDT_AixControllerStatus";
      END_STRUCT;
      "730" : Struct
         Conveyor { S7_SetPoint := 'False'} : "UDT_ConveyorStatus";
         PEC_EoS : "UDT_PECStatus";
         MCO_M01 { S7_SetPoint := 'False'} : "UDT_AixControllerStatus";
      END_STRUCT;
      "740" : Struct
         Conveyor { S7_SetPoint := 'False'} : "UDT_ConveyorStatus";
         PEC_EoS { S7_SetPoint := 'False'} : "UDT_PECStatus";
         MCO_M01 : "UDT_AixControllerStatus";
      END_STRUCT;
      "750" : Struct
         Conveyor { S7_SetPoint := 'False'} : "UDT_ConveyorStatus";
         PEC_EoS : "UDT_PECStatus";
         MCO_M01 { S7_SetPoint := 'False'} : "UDT_AixControllerStatus";
      END_STRUCT;
   END_STRUCT;

END_TYPE

TYPE "UDT_WSGStatistics"
VERSION : 0.1
   STRUCT
      "010" : Struct
         Conveyor { S7_SetPoint := 'False'} : "UDT_ConveyorStatistics";
         PEC_EoS : "UDT_PECStatistics";
         MCO_M01 : "UDT_VfdStatistics";
      END_STRUCT;
      "020" : Struct
         Conveyor { S7_SetPoint := 'False'} : "UDT_ConveyorStatistics";
         PEC_EoS : "UDT_PECStatistics";
         MCO_M01 { S7_SetPoint := 'False'} : "UDT_VfdStatistics";
      END_STRUCT;
      "021" : Struct
         RightAngledTransfer { S7_SetPoint := 'False'} : "UDT_RATStatistics";
         MCO_M01 : "UDT_VfdStatistics";
      END_STRUCT;
      "110" : Struct
         Conveyor { S7_SetPoint := 'False'} : "UDT_ConveyorStatistics";
         PEC_EoS : "UDT_PECUpdateStatistics";
         MCO_M01 { S7_SetPoint := 'False'} : "UDT_VfdStatistics";
      END_STRUCT;
      "120" : Struct
         Conveyor { S7_SetPoint := 'False'} : "UDT_ConveyorStatistics";
         PEC_EoS : "UDT_PECStatistics";
         MCO_M01 : "UDT_VfdStatistics";
      END_STRUCT;
      "130" : Struct
         Conveyor { S7_SetPoint := 'False'} : "UDT_ConveyorStatistics";
         PEC_EoS : "UDT_PECUpdateStatistics";
         MCO_M01 : "UDT_VfdStatistics";
      END_STRUCT;
      "140" : Struct
         Conveyor { S7_SetPoint := 'False'} : "UDT_ConveyorStatistics";
         PEC_EoS : "UDT_PECStatistics";
         MCO_M01 { S7_SetPoint := 'False'} : "UDT_VfdStatistics";
      END_STRUCT;
      "141" : Struct
         RightAngledTransfer { S7_SetPoint := 'False'} : "UDT_RATStatistics";
         MCO_M01 : "UDT_VfdStatistics";
      END_STRUCT;
      "150" : Struct
         Conveyor { S7_SetPoint := 'False'} : "UDT_ConveyorStatistics";
         PEC_EoS : "UDT_PECUpdateStatistics";
         MCO_M01 { S7_SetPoint := 'False'} : "UDT_VfdStatistics";
      END_STRUCT;
      "160" : Struct
         Conveyor { S7_SetPoint := 'False'} : "UDT_ConveyorStatistics";
         PEC_EoS : "UDT_PECUpdateStatistics";
         MCO_M01 : "UDT_VfdStatistics";
      END_STRUCT;
      "170" : Struct
         Conveyor { S7_SetPoint := 'False'} : "UDT_ConveyorStatistics";
         PEC_EoS : "UDT_PECUpdateStatistics";
         MCO_M01 { S7_SetPoint := 'False'} : "UDT_VfdStatistics";
      END_STRUCT;
      "180" : Struct
         Conveyor { S7_SetPoint := 'False'} : "UDT_ConveyorStatistics";
         PEC_EoS : "UDT_PECUpdateStatistics";
         MCO_M01 : "UDT_VfdStatistics";
      END_STRUCT;
      "190" : Struct
         Conveyor { S7_SetPoint := 'False'} : "UDT_ConveyorStatistics";
         PEC_EoS : "UDT_PECUpdateStatistics";
         MCO_M01 { S7_SetPoint := 'False'} : "UDT_VfdStatistics";
      END_STRUCT;
      "210" : Struct
         Conveyor { S7_SetPoint := 'False'} : "UDT_ConveyorStatistics";
         PEC_EoS : "UDT_PECStatistics";
         MCO_M01 { S7_SetPoint := 'False'} : "UDT_VfdStatistics";
      END_STRUCT;
      "211" : Struct
         RightAngledTransfer { S7_SetPoint := 'False'} : "UDT_RATStatistics";
         MCO_M01 : "UDT_VfdStatistics";
      END_STRUCT;
      "220" : Struct
         Conveyor { S7_SetPoint := 'False'} : "UDT_ConveyorStatistics";
         PEC_EoS : "UDT_PECStatistics";
         MCO_M01 { S7_SetPoint := 'False'} : "UDT_VfdStatistics";
      END_STRUCT;
      "221" : Struct
         RightAngledTransfer { S7_SetPoint := 'False'} : "UDT_RATStatistics";
         MCO_M01 : "UDT_VfdStatistics";
      END_STRUCT;
      "230" : Struct
         Conveyor { S7_SetPoint := 'False'} : "UDT_ConveyorStatistics";
         MCO_M01 { S7_SetPoint := 'False'} : "UDT_VfdStatistics";
      END_STRUCT;
      "310" : Struct
         Conveyor { S7_SetPoint := 'False'} : "UDT_ConveyorStatistics";
         PEC_EoS : "UDT_PECStatistics";
         MCO_M01 { S7_SetPoint := 'False'} : "UDT_VfdStatistics";
      END_STRUCT;
      "320" : Struct
         Conveyor { S7_SetPoint := 'False'} : "UDT_ConveyorStatistics";
         PEC_EoS : "UDT_PECStatistics";
         MCO_M01 : "UDT_VfdStatistics";
      END_STRUCT;
      "330" : Struct
         Conveyor { S7_SetPoint := 'False'} : "UDT_ConveyorStatistics";
         PEC_EoS : "UDT_PECStatistics";
         MCO_M01 { S7_SetPoint := 'False'} : "UDT_VfdStatistics";
      END_STRUCT;
      "340" : Struct
         Conveyor { S7_SetPoint := 'False'} : "UDT_ConveyorStatistics";
         PEC_EoS : "UDT_PECStatistics";
         MCO_M01 : "UDT_VfdStatistics";
      END_STRUCT;
      "350" : Struct
         Conveyor { S7_SetPoint := 'False'} : "UDT_ConveyorStatistics";
         PEC_EoS : "UDT_PECStatistics";
         MCO_M01 { S7_SetPoint := 'False'} : "UDT_VfdStatistics";
      END_STRUCT;
      "510" : Struct
         Conveyor { S7_SetPoint := 'False'} : "UDT_ConveyorStatistics";
         MCO_M01 { S7_SetPoint := 'False'} : "UDT_VfdStatistics";
      END_STRUCT;
      "520" : Struct
         Conveyor { S7_SetPoint := 'False'} : "UDT_ConveyorStatistics";
         PEC_EoS : "UDT_PECUpdateStatistics";
         MCO_M01 { S7_SetPoint := 'False'} : "UDT_VfdStatistics";
      END_STRUCT;
      "530" : Struct
         Conveyor { S7_SetPoint := 'False'} : "UDT_ConveyorStatistics";
         PEC_EoS : "UDT_PECUpdateStatistics";
         MCO_M01 : "UDT_VfdStatistics";
      END_STRUCT;
      "540" : Struct
         Conveyor { S7_SetPoint := 'False'} : "UDT_ConveyorStatistics";
         PEC_EoS : "UDT_PECStatistics";
         MCO_M01 { S7_SetPoint := 'False'} : "UDT_VfdStatistics";
      END_STRUCT;
      "541" : Struct
         RightAngledTransfer { S7_SetPoint := 'False'} : "UDT_RATStatistics";
         MCO_M01 : "UDT_VfdStatistics";
      END_STRUCT;
      "550" : Struct
         Conveyor { S7_SetPoint := 'False'} : "UDT_ConveyorStatistics";
         PEC_EoS : "UDT_PECUpdateStatistics";
         MCO_M01 { S7_SetPoint := 'False'} : "UDT_VfdStatistics";
      END_STRUCT;
      "560" : Struct
         Conveyor { S7_SetPoint := 'False'} : "UDT_ConveyorStatistics";
         PEC_EoS : "UDT_PECUpdateStatistics";
         MCO_M01 : "UDT_VfdStatistics";
      END_STRUCT;
      "570" : Struct
         Conveyor { S7_SetPoint := 'False'} : "UDT_ConveyorStatistics";
         PEC_EoS : "UDT_PECUpdateStatistics";
         MCO_M01 { S7_SetPoint := 'False'} : "UDT_VfdStatistics";
      END_STRUCT;
      "580" : Struct
         Conveyor { S7_SetPoint := 'False'} : "UDT_ConveyorStatistics";
         PEC_EoS : "UDT_PECUpdateStatistics";
         MCO_M01 : "UDT_VfdStatistics";
      END_STRUCT;
      "590" : Struct
         Conveyor { S7_SetPoint := 'False'} : "UDT_ConveyorStatistics";
         PEC_EoS : "UDT_PECUpdateStatistics";
         MCO_M01 { S7_SetPoint := 'False'} : "UDT_VfdStatistics";
      END_STRUCT;
      "610" : Struct
         Conveyor { S7_SetPoint := 'False'} : "UDT_ConveyorStatistics";
         PEC_EoS : "UDT_PECStatistics";
         MCO_M01 { S7_SetPoint := 'False'} : "UDT_VfdStatistics";
      END_STRUCT;
      "611" : Struct
         RightAngledTransfer { S7_SetPoint := 'False'} : "UDT_RATStatistics";
         MCO_M01 : "UDT_VfdStatistics";
      END_STRUCT;
      "620" : Struct
         Conveyor { S7_SetPoint := 'False'} : "UDT_ConveyorStatistics";
         PEC_EoS : "UDT_PECStatistics";
         MCO_M01 { S7_SetPoint := 'False'} : "UDT_VfdStatistics";
      END_STRUCT;
      "621" : Struct
         RightAngledTransfer { S7_SetPoint := 'False'} : "UDT_RATStatistics";
         MCO_M01 : "UDT_VfdStatistics";
      END_STRUCT;
      "630" : Struct
         Conveyor { S7_SetPoint := 'False'} : "UDT_ConveyorStatistics";
         MCO_M01 { S7_SetPoint := 'False'} : "UDT_VfdStatistics";
      END_STRUCT;
      "710" : Struct
         Conveyor { S7_SetPoint := 'False'} : "UDT_ConveyorStatistics";
         PEC_EoS : "UDT_PECStatistics";
         MCO_M01 { S7_SetPoint := 'False'} : "UDT_VfdStatistics";
      END_STRUCT;
      "720" : Struct
         Conveyor { S7_SetPoint := 'False'} : "UDT_ConveyorStatistics";
         PEC_EoS : "UDT_PECStatistics";
         MCO_M01 : "UDT_VfdStatistics";
      END_STRUCT;
      "730" : Struct
         Conveyor { S7_SetPoint := 'False'} : "UDT_ConveyorStatistics";
         PEC_EoS : "UDT_PECStatistics";
         MCO_M01 { S7_SetPoint := 'False'} : "UDT_VfdStatistics";
      END_STRUCT;
      "740" : Struct
         Conveyor { S7_SetPoint := 'False'} : "UDT_ConveyorStatistics";
         PEC_EoS : "UDT_PECStatistics";
         MCO_M01 : "UDT_VfdStatistics";
      END_STRUCT;
      "750" : Struct
         Conveyor { S7_SetPoint := 'False'} : "UDT_ConveyorStatistics";
         PEC_EoS : "UDT_PECStatistics";
         MCO_M01 { S7_SetPoint := 'False'} : "UDT_VfdStatistics";
      END_STRUCT;
   END_STRUCT;

END_TYPE

TYPE "UDT_WSGHmiCommands"
VERSION : 0.1
   STRUCT
      "010" { ExternalAccessible := 'False'; ExternalVisible := 'False'; ExternalWritable := 'False'} : Struct
         Conveyor { ExternalAccessible := 'False'; ExternalVisible := 'False'; ExternalWritable := 'False'; S7_SetPoint := 'False'} : "UDT_ConveyorCommand";
      END_STRUCT;
      "020" { ExternalAccessible := 'False'; ExternalVisible := 'False'; ExternalWritable := 'False'} : Struct
         Conveyor { ExternalAccessible := 'False'; ExternalVisible := 'False'; ExternalWritable := 'False'; S7_SetPoint := 'False'} : "UDT_ConveyorCommand";
      END_STRUCT;
      "021" { ExternalAccessible := 'False'; ExternalVisible := 'False'; ExternalWritable := 'False'} : Struct
         RAT { ExternalAccessible := 'False'; ExternalVisible := 'False'; ExternalWritable := 'False'; S7_SetPoint := 'False'} : "UDT_RATCommand";
      END_STRUCT;
      "110" { ExternalAccessible := 'False'; ExternalVisible := 'False'; ExternalWritable := 'False'} : Struct
         Conveyor { ExternalAccessible := 'False'; ExternalVisible := 'False'; ExternalWritable := 'False'; S7_SetPoint := 'False'} : "UDT_ConveyorCommand";
      END_STRUCT;
      "120" { ExternalAccessible := 'False'; ExternalVisible := 'False'; ExternalWritable := 'False'} : Struct
         Conveyor { ExternalAccessible := 'False'; ExternalVisible := 'False'; ExternalWritable := 'False'; S7_SetPoint := 'False'} : "UDT_ConveyorCommand";
      END_STRUCT;
      "130" { ExternalAccessible := 'False'; ExternalVisible := 'False'; ExternalWritable := 'False'} : Struct
         Conveyor { ExternalAccessible := 'False'; ExternalVisible := 'False'; ExternalWritable := 'False'; S7_SetPoint := 'False'} : "UDT_ConveyorCommand";
      END_STRUCT;
      "140" { ExternalAccessible := 'False'; ExternalVisible := 'False'; ExternalWritable := 'False'} : Struct
         Conveyor { ExternalAccessible := 'False'; ExternalVisible := 'False'; ExternalWritable := 'False'; S7_SetPoint := 'False'} : "UDT_ConveyorCommand";
      END_STRUCT;
      "141" { ExternalAccessible := 'False'; ExternalVisible := 'False'; ExternalWritable := 'False'} : Struct
         RightAngledTransfer { ExternalAccessible := 'False'; ExternalVisible := 'False'; ExternalWritable := 'False'; S7_SetPoint := 'False'} : "UDT_RATCommand";
      END_STRUCT;
      "150" { ExternalAccessible := 'False'; ExternalVisible := 'False'; ExternalWritable := 'False'} : Struct
         Conveyor { ExternalAccessible := 'False'; ExternalVisible := 'False'; ExternalWritable := 'False'; S7_SetPoint := 'False'} : "UDT_ConveyorCommand";
      END_STRUCT;
      "160" { ExternalAccessible := 'False'; ExternalVisible := 'False'; ExternalWritable := 'False'} : Struct
         Conveyor { ExternalAccessible := 'False'; ExternalVisible := 'False'; ExternalWritable := 'False'; S7_SetPoint := 'False'} : "UDT_ConveyorCommand";
      END_STRUCT;
      "170" { ExternalAccessible := 'False'; ExternalVisible := 'False'; ExternalWritable := 'False'} : Struct
         Conveyor { ExternalAccessible := 'False'; ExternalVisible := 'False'; ExternalWritable := 'False'; S7_SetPoint := 'False'} : "UDT_ConveyorCommand";
      END_STRUCT;
      "180" { ExternalAccessible := 'False'; ExternalVisible := 'False'; ExternalWritable := 'False'} : Struct
         Conveyor { ExternalAccessible := 'False'; ExternalVisible := 'False'; ExternalWritable := 'False'; S7_SetPoint := 'False'} : "UDT_ConveyorCommand";
      END_STRUCT;
      "190" { ExternalAccessible := 'False'; ExternalVisible := 'False'; ExternalWritable := 'False'} : Struct
         Conveyor { ExternalAccessible := 'False'; ExternalVisible := 'False'; ExternalWritable := 'False'; S7_SetPoint := 'False'} : "UDT_ConveyorCommand";
      END_STRUCT;
      "210" { ExternalAccessible := 'False'; ExternalVisible := 'False'; ExternalWritable := 'False'} : Struct
         Conveyor { ExternalAccessible := 'False'; ExternalVisible := 'False'; ExternalWritable := 'False'; S7_SetPoint := 'False'} : "UDT_ConveyorCommand";
      END_STRUCT;
      "211" { ExternalAccessible := 'False'; ExternalVisible := 'False'; ExternalWritable := 'False'} : Struct
         RightAngledTransfer { ExternalAccessible := 'False'; ExternalVisible := 'False'; ExternalWritable := 'False'; S7_SetPoint := 'False'} : "UDT_RATCommand";
      END_STRUCT;
      "220" { ExternalAccessible := 'False'; ExternalVisible := 'False'; ExternalWritable := 'False'} : Struct
         Conveyor { ExternalAccessible := 'False'; ExternalVisible := 'False'; ExternalWritable := 'False'; S7_SetPoint := 'False'} : "UDT_ConveyorCommand";
      END_STRUCT;
      "221" { ExternalAccessible := 'False'; ExternalVisible := 'False'; ExternalWritable := 'False'} : Struct
         RightAngledTransfer { ExternalAccessible := 'False'; ExternalVisible := 'False'; ExternalWritable := 'False'; S7_SetPoint := 'False'} : "UDT_RATCommand";
      END_STRUCT;
      "230" { ExternalAccessible := 'False'; ExternalVisible := 'False'; ExternalWritable := 'False'} : Struct
         Conveyor { ExternalAccessible := 'False'; ExternalVisible := 'False'; ExternalWritable := 'False'; S7_SetPoint := 'False'} : "UDT_ConveyorCommand";
      END_STRUCT;
      "310" { ExternalAccessible := 'False'; ExternalVisible := 'False'; ExternalWritable := 'False'} : Struct
         Conveyor { ExternalAccessible := 'False'; ExternalVisible := 'False'; ExternalWritable := 'False'; S7_SetPoint := 'False'} : "UDT_ConveyorCommand";
      END_STRUCT;
      "320" { ExternalAccessible := 'False'; ExternalVisible := 'False'; ExternalWritable := 'False'} : Struct
         Conveyor { ExternalAccessible := 'False'; ExternalVisible := 'False'; ExternalWritable := 'False'; S7_SetPoint := 'False'} : "UDT_ConveyorCommand";
      END_STRUCT;
      "330" { ExternalAccessible := 'False'; ExternalVisible := 'False'; ExternalWritable := 'False'} : Struct
         Conveyor { ExternalAccessible := 'False'; ExternalVisible := 'False'; ExternalWritable := 'False'; S7_SetPoint := 'False'} : "UDT_ConveyorCommand";
      END_STRUCT;
      "340" { ExternalAccessible := 'False'; ExternalVisible := 'False'; ExternalWritable := 'False'} : Struct
         Conveyor { ExternalAccessible := 'False'; ExternalVisible := 'False'; ExternalWritable := 'False'; S7_SetPoint := 'False'} : "UDT_ConveyorCommand";
      END_STRUCT;
      "350" { ExternalAccessible := 'False'; ExternalVisible := 'False'; ExternalWritable := 'False'} : Struct
         Conveyor { ExternalAccessible := 'False'; ExternalVisible := 'False'; ExternalWritable := 'False'; S7_SetPoint := 'False'} : "UDT_ConveyorCommand";
      END_STRUCT;
      "510" { ExternalAccessible := 'False'; ExternalVisible := 'False'; ExternalWritable := 'False'} : Struct
         Conveyor { ExternalAccessible := 'False'; ExternalVisible := 'False'; ExternalWritable := 'False'; S7_SetPoint := 'False'} : "UDT_ConveyorCommand";
      END_STRUCT;
      "520" { ExternalAccessible := 'False'; ExternalVisible := 'False'; ExternalWritable := 'False'} : Struct
         Conveyor { ExternalAccessible := 'False'; ExternalVisible := 'False'; ExternalWritable := 'False'; S7_SetPoint := 'False'} : "UDT_ConveyorCommand";
      END_STRUCT;
      "530" { ExternalAccessible := 'False'; ExternalVisible := 'False'; ExternalWritable := 'False'} : Struct
         Conveyor { ExternalAccessible := 'False'; ExternalVisible := 'False'; ExternalWritable := 'False'; S7_SetPoint := 'False'} : "UDT_ConveyorCommand";
      END_STRUCT;
      "540" { ExternalAccessible := 'False'; ExternalVisible := 'False'; ExternalWritable := 'False'} : Struct
         Conveyor { ExternalAccessible := 'False'; ExternalVisible := 'False'; ExternalWritable := 'False'; S7_SetPoint := 'False'} : "UDT_ConveyorCommand";
      END_STRUCT;
      "541" { ExternalAccessible := 'False'; ExternalVisible := 'False'; ExternalWritable := 'False'} : Struct
         RightAngledTransfer { ExternalAccessible := 'False'; ExternalVisible := 'False'; ExternalWritable := 'False'; S7_SetPoint := 'False'} : "UDT_RATCommand";
      END_STRUCT;
      "550" { ExternalAccessible := 'False'; ExternalVisible := 'False'; ExternalWritable := 'False'} : Struct
         Conveyor { ExternalAccessible := 'False'; ExternalVisible := 'False'; ExternalWritable := 'False'; S7_SetPoint := 'False'} : "UDT_ConveyorCommand";
      END_STRUCT;
      "560" { ExternalAccessible := 'False'; ExternalVisible := 'False'; ExternalWritable := 'False'} : Struct
         Conveyor { ExternalAccessible := 'False'; ExternalVisible := 'False'; ExternalWritable := 'False'; S7_SetPoint := 'False'} : "UDT_ConveyorCommand";
      END_STRUCT;
      "570" { ExternalAccessible := 'False'; ExternalVisible := 'False'; ExternalWritable := 'False'} : Struct
         Conveyor { ExternalAccessible := 'False'; ExternalVisible := 'False'; ExternalWritable := 'False'; S7_SetPoint := 'False'} : "UDT_ConveyorCommand";
      END_STRUCT;
      "580" { ExternalAccessible := 'False'; ExternalVisible := 'False'; ExternalWritable := 'False'} : Struct
         Conveyor { ExternalAccessible := 'False'; ExternalVisible := 'False'; ExternalWritable := 'False'; S7_SetPoint := 'False'} : "UDT_ConveyorCommand";
      END_STRUCT;
      "590" { ExternalAccessible := 'False'; ExternalVisible := 'False'; ExternalWritable := 'False'} : Struct
         Conveyor { ExternalAccessible := 'False'; ExternalVisible := 'False'; ExternalWritable := 'False'; S7_SetPoint := 'False'} : "UDT_ConveyorCommand";
      END_STRUCT;
      "610" { ExternalAccessible := 'False'; ExternalVisible := 'False'; ExternalWritable := 'False'} : Struct
         Conveyor { ExternalAccessible := 'False'; ExternalVisible := 'False'; ExternalWritable := 'False'; S7_SetPoint := 'False'} : "UDT_ConveyorCommand";
      END_STRUCT;
      "611" { ExternalAccessible := 'False'; ExternalVisible := 'False'; ExternalWritable := 'False'} : Struct
         RightAngledTransfer { ExternalAccessible := 'False'; ExternalVisible := 'False'; ExternalWritable := 'False'; S7_SetPoint := 'False'} : "UDT_RATCommand";
      END_STRUCT;
      "620" { ExternalAccessible := 'False'; ExternalVisible := 'False'; ExternalWritable := 'False'} : Struct
         Conveyor { ExternalAccessible := 'False'; ExternalVisible := 'False'; ExternalWritable := 'False'; S7_SetPoint := 'False'} : "UDT_ConveyorCommand";
      END_STRUCT;
      "621" { ExternalAccessible := 'False'; ExternalVisible := 'False'; ExternalWritable := 'False'} : Struct
         RightAngledTransfer { ExternalAccessible := 'False'; ExternalVisible := 'False'; ExternalWritable := 'False'; S7_SetPoint := 'False'} : "UDT_RATCommand";
      END_STRUCT;
      "630" { ExternalAccessible := 'False'; ExternalVisible := 'False'; ExternalWritable := 'False'} : Struct
         Conveyor { ExternalAccessible := 'False'; ExternalVisible := 'False'; ExternalWritable := 'False'; S7_SetPoint := 'False'} : "UDT_ConveyorCommand";
      END_STRUCT;
      "710" { ExternalAccessible := 'False'; ExternalVisible := 'False'; ExternalWritable := 'False'} : Struct
         Conveyor { ExternalAccessible := 'False'; ExternalVisible := 'False'; ExternalWritable := 'False'; S7_SetPoint := 'False'} : "UDT_ConveyorCommand";
      END_STRUCT;
      "720" { ExternalAccessible := 'False'; ExternalVisible := 'False'; ExternalWritable := 'False'} : Struct
         Conveyor { ExternalAccessible := 'False'; ExternalVisible := 'False'; ExternalWritable := 'False'; S7_SetPoint := 'False'} : "UDT_ConveyorCommand";
      END_STRUCT;
      "730" { ExternalAccessible := 'False'; ExternalVisible := 'False'; ExternalWritable := 'False'} : Struct
         Conveyor { ExternalAccessible := 'False'; ExternalVisible := 'False'; ExternalWritable := 'False'; S7_SetPoint := 'False'} : "UDT_ConveyorCommand";
      END_STRUCT;
      "740" { ExternalAccessible := 'False'; ExternalVisible := 'False'; ExternalWritable := 'False'} : Struct
         Conveyor { ExternalAccessible := 'False'; ExternalVisible := 'False'; ExternalWritable := 'False'; S7_SetPoint := 'False'} : "UDT_ConveyorCommand";
      END_STRUCT;
      "750" { ExternalAccessible := 'False'; ExternalVisible := 'False'; ExternalWritable := 'False'} : Struct
         Conveyor { ExternalAccessible := 'False'; ExternalVisible := 'False'; ExternalWritable := 'False'; S7_SetPoint := 'False'} : "UDT_ConveyorCommand";
      END_STRUCT;
   END_STRUCT;

END_TYPE

TYPE "UDT_NerakLiftStatus"
VERSION : 0.1
   STRUCT
      Status : Int;   // Status number
      Specific : Struct
         Reverse : Bool;
         CollisionDetected : Bool;
         ProductFellDown : Bool;
      END_STRUCT;
   END_STRUCT;

END_TYPE

TYPE "UDT_WSRStatistics"
VERSION : 0.1
   STRUCT
      "010" { S7_SetPoint := 'False'} : "UDT_StatisticsTC03";
      "020" { S7_SetPoint := 'False'} : "UDT_StatisticsTC13";
      "030" { S7_SetPoint := 'False'} : "UDT_StatisticsTC03";
      "040" { S7_SetPoint := 'False'} : "UDT_StatisticsTC07";
      "041" { S7_SetPoint := 'False'} : "UDT_StatisticsTC36";
      "050" { S7_SetPoint := 'False'} : "UDT_StatisticsTC03";
      "060" { S7_SetPoint := 'False'} : "UDT_StatisticsTC13";
      "070" { S7_SetPoint := 'False'} : "UDT_StatisticsTC03";
      "080" { S7_SetPoint := 'False'} : "UDT_StatisticsTC13";
      "110" { S7_SetPoint := 'False'} : "UDT_StatisticsTC03";
      "120" { S7_SetPoint := 'False'} : "UDT_StatisticsTC13";
      "130" { S7_SetPoint := 'False'} : "UDT_StatisticsTC03";
      "140" { S7_SetPoint := 'False'} : "UDT_StatisticsTC07";
      "141" { S7_SetPoint := 'False'} : "UDT_StatisticsTC36";
      "150" { S7_SetPoint := 'False'} : "UDT_StatisticsTC03";
      "160" { S7_SetPoint := 'False'} : "UDT_StatisticsTC13";
      "170" { S7_SetPoint := 'False'} : "UDT_StatisticsTC03";
      "180" { S7_SetPoint := 'False'} : "UDT_StatisticsTC11";
      "210" { S7_SetPoint := 'False'} : "UDT_StatisticsTC03";
      "220" { S7_SetPoint := 'False'} : "UDT_StatisticsTC13";
      "230" { S7_SetPoint := 'False'} : "UDT_StatisticsTC03";
      "240" { S7_SetPoint := 'False'} : "UDT_StatisticsTC02";
      "241" { S7_SetPoint := 'False'} : "UDT_StatisticsTC36";
      "250" { S7_SetPoint := 'False'} : "UDT_StatisticsTC03";
      "260" { S7_SetPoint := 'False'} : "UDT_StatisticsTC13";
      "270" { S7_SetPoint := 'False'} : "UDT_StatisticsTC03";
   END_STRUCT;

END_TYPE

TYPE "UDT_ScannerInterface"
VERSION : 0.1
   STRUCT
      Trigger : Bool;
      BarCodeValue : String;
   END_STRUCT;

END_TYPE

FUNCTION_BLOCK "FB_DataLogicBladeSN"
{ S7_Optimized_Access := 'TRUE' }
VERSION : 0.1
   VAR_INPUT
      iudt_DataLogicBladeIN { ExternalAccessible := 'False'; ExternalVisible := 'False'; ExternalWritable := 'False'} : "UDT_DataLogicBlade_IN_SN";
      ix_Trigger { ExternalAccessible := 'False'; ExternalVisible := 'False'; ExternalWritable := 'False'} : Bool;
   END_VAR

   VAR_OUTPUT
      qx_Trigger { ExternalAccessible := 'False'; ExternalVisible := 'False'; ExternalWritable := 'False'} : Bool;
      qs_Barcode { ExternalAccessible := 'False'; ExternalVisible := 'False'; ExternalWritable := 'False'} : String;
   END_VAR

   VAR
      sa_Data { ExternalAccessible := 'False'; ExternalVisible := 'False'; ExternalWritable := 'False'} : Array[0..14] of Char;
      R_TRIG_Trigger {InstructionName := 'R_TRIG'; LibVersion := '1.0'; ExternalAccessible := 'False'; ExternalVisible := 'False'; ExternalWritable := 'False'; S7_SetPoint := 'False'} : R_TRIG;   // Rising edge trigger signal
      R_TRIG_Succes {InstructionName := 'R_TRIG'; LibVersion := '1.0'; ExternalAccessible := 'False'; ExternalVisible := 'False'; ExternalWritable := 'False'; S7_SetPoint := 'False'} : R_TRIG;
      R_TRIG_Failure {InstructionName := 'R_TRIG'; LibVersion := '1.0'; ExternalAccessible := 'False'; ExternalVisible := 'False'; ExternalWritable := 'False'; S7_SetPoint := 'False'} : R_TRIG;
      sfb_TimerOnOffDelay_Trigger { ExternalAccessible := 'False'; ExternalVisible := 'False'; ExternalWritable := 'False'; S7_SetPoint := 'False'} : "FB_TimerOnOffDelay";
      si_Index { ExternalAccessible := 'False'; ExternalVisible := 'False'; ExternalWritable := 'False'} : Int;
      si_GoodReadCount { ExternalAccessible := 'False'; ExternalVisible := 'False'; ExternalWritable := 'False'} : Int;
      si_BadReadCount { ExternalAccessible := 'False'; ExternalVisible := 'False'; ExternalWritable := 'False'} : Int;
      sx_Trigger { ExternalAccessible := 'False'; ExternalVisible := 'False'; ExternalWritable := 'False'} : Bool;
   END_VAR


BEGIN
	#R_TRIG_Trigger(CLK := #ix_Trigger);  //Rising edge trigger signal
	#R_TRIG_Succes(CLK := #iudt_DataLogicBladeIN.Data[0].%X0);//AND NOT #sx_Trigger);
	#R_TRIG_Failure(CLK := #iudt_DataLogicBladeIN.Data[0].%X1);// AND NOT #sx_Trigger);

	REGION 1 - Scanning
	    IF #R_TRIG_Trigger.Q THEN
	        #sx_Trigger := TRUE;
	    END_IF;

	    #sfb_TimerOnOffDelay_Trigger(iudi_OnDelayTime := 600,
	                                 ix_SignalToDelay := #sx_Trigger,
	                                 ix_Enable := TRUE);

	    IF #sfb_TimerOnOffDelay_Trigger.qx_DelayedSignal THEN
	        #sx_Trigger := FALSE;
	    END_IF;




	    IF #R_TRIG_Succes.Q OR #R_TRIG_Failure.Q THEN

	        FOR #si_Index := 1 TO 15 DO
	            #sa_Data[#si_Index - 1] := BYTE_TO_CHAR(#iudt_DataLogicBladeIN.Data[#si_Index]);
	        END_FOR;

	        IF #sa_Data[0] = '$02' AND #sa_Data[11] = '$R' AND #sa_Data[12] = '$L' THEN
	            Chars_TO_Strg(Chars := #sa_Data,
	                          pChars := 1,
	                          Cnt := 10,
	                          Strg => #qs_Barcode);
	            #si_GoodReadCount += 1;

	        ELSIF #sa_Data[1] = '$18' THEN
	            #qs_Barcode := 'NO_READ    ';
	            #si_BadReadCount += 1;

	        END_IF;


	    END_IF;
	END_REGION


	REGION 2 - Output write
	    #qx_Trigger := #sx_Trigger;
	END_REGION




END_FUNCTION_BLOCK

TYPE "UDT_TGWLiftPO"
VERSION : 0.1
   STRUCT
      qx_Fault : Bool;   // Fault lamp
      qx_MainContactorOn : Bool;   // Main contactor on
      Spare_1 : Bool;
      Spare_2 : Bool;
      Spare_3 : Bool;
      Spare_4 : Bool;
      Spare_5 : Bool;
      Spare_6 : Bool;
   END_STRUCT;

END_TYPE

FUNCTION_BLOCK "FB_LiftManualControl"
{ S7_Optimized_Access := 'TRUE' }
VERSION : 0.1
// ATTRIBUTES
// AUTO_NUMBER = True
// BLOCK_NUMBER = 263
// END_ATTRIBUTES
   VAR_INPUT
      ix_ManualMode { ExternalAccessible := 'False'; ExternalVisible := 'False'; ExternalWritable := 'False'} : Bool;
      ix_AutoMode { ExternalAccessible := 'False'; ExternalVisible := 'False'; ExternalWritable := 'False'} : Bool;
      ix_UpPosition { ExternalAccessible := 'False'; ExternalVisible := 'False'; ExternalWritable := 'False'} : Bool;
      ix_DownPosition { ExternalAccessible := 'False'; ExternalVisible := 'False'; ExternalWritable := 'False'} : Bool;
      ix_LiftConveyorRight { ExternalAccessible := 'False'; ExternalVisible := 'False'; ExternalWritable := 'False'} : Bool;
      ix_LiftConveyorLeft { ExternalAccessible := 'False'; ExternalVisible := 'False'; ExternalWritable := 'False'} : Bool;
      ix_InfeedConveyor { ExternalAccessible := 'False'; ExternalVisible := 'False'; ExternalWritable := 'False'} : Bool;
      ix_OutfeedConveyor { ExternalAccessible := 'False'; ExternalVisible := 'False'; ExternalWritable := 'False'} : Bool;
   END_VAR

   VAR_IN_OUT
      iqUDT_LiftConveyorCommand : "UDT_ConveyorCommand";
      iqUDT_LowerInfeedConveyorCommand : "UDT_ConveyorCommand";
      iqUDT_LowerOutfeedConveyorCommand : "UDT_ConveyorCommand";
      iqUDT_UpperInfeedConveyorCommand : "UDT_ConveyorCommand";
      iqUDT_UpperOutfeedConveyorCommand : "UDT_ConveyorCommand";
   END_VAR


BEGIN
	(*

	----------------------------------------------------------------------------------------

	Version history:
	Date        | Version   | Author        | Remark
	----------------------------------------------------------------------------------------
	14/06/2024  | 1.0       | R.Pieczonka   | First release
	*)

	REGION Modes
	    //Setting manual mode for lift, infeed and outfeed conveyors if key-operated switch is turned to manual mode
	    IF #ix_ManualMode THEN
	        #iqUDT_LiftConveyorCommand.ManualMode := TRUE;
	        #iqUDT_LowerInfeedConveyorCommand.ManualMode := TRUE;
	        #iqUDT_LowerOutfeedConveyorCommand.ManualMode := TRUE;
	        #iqUDT_UpperInfeedConveyorCommand.ManualMode := TRUE;
	        #iqUDT_UpperOutfeedConveyorCommand.ManualMode := TRUE;
	    END_IF;

	    //Setting automatic mode for lift, infeed and outfeed conveyors if key-operated switch is turned to automatic mode
	    IF #ix_AutoMode THEN
	        #iqUDT_LiftConveyorCommand.ManualMode := FALSE;
	        #iqUDT_LowerInfeedConveyorCommand.ManualMode := FALSE;
	        #iqUDT_LowerOutfeedConveyorCommand.ManualMode := FALSE;
	        #iqUDT_UpperInfeedConveyorCommand.ManualMode := FALSE;
	        #iqUDT_UpperOutfeedConveyorCommand.ManualMode := FALSE;
	    END_IF;
	END_REGION

	REGION Lift Conveyor
	    //Commands for controling only lift conveyor
	    IF #iqUDT_LiftConveyorCommand.ManualMode AND #ix_LiftConveyorRight THEN
	        #iqUDT_LiftConveyorCommand.ManualStartStop := TRUE;
	        #iqUDT_LiftConveyorCommand.Reverse := FALSE;

	    ELSIF #iqUDT_LiftConveyorCommand.ManualMode AND #ix_LiftConveyorLeft THEN
	        #iqUDT_LiftConveyorCommand.ManualStartStop := TRUE;
	        #iqUDT_LiftConveyorCommand.Reverse := TRUE;
	    ELSE
	        #iqUDT_LiftConveyorCommand.ManualStartStop := FALSE;
	        #iqUDT_LiftConveyorCommand.Reverse := FALSE;
	    END_IF;
	END_REGION

	REGION Lower Position
	    //Lower infeed
	    IF #iqUDT_LiftConveyorCommand.ManualMode
	        AND #iqUDT_LowerInfeedConveyorCommand.ManualMode
	        AND #ix_DownPosition
	        AND #ix_LiftConveyorRight
	        AND #ix_InfeedConveyor
	    THEN
	        #iqUDT_LiftConveyorCommand.ManualStartStop := TRUE;
	        #iqUDT_LiftConveyorCommand.Reverse := FALSE;
	        #iqUDT_LowerInfeedConveyorCommand.ManualStartStop := TRUE;
	        #iqUDT_LowerInfeedConveyorCommand.Reverse := FALSE;

	    ELSIF #iqUDT_LiftConveyorCommand.ManualMode
	        AND #iqUDT_LowerInfeedConveyorCommand.ManualMode
	        AND #ix_DownPosition
	        AND #ix_LiftConveyorLeft
	        AND #ix_InfeedConveyor
	    THEN
	        #iqUDT_LiftConveyorCommand.ManualStartStop := TRUE;
	        #iqUDT_LiftConveyorCommand.Reverse := TRUE;
	        #iqUDT_LowerInfeedConveyorCommand.ManualStartStop := TRUE;
	        #iqUDT_LowerInfeedConveyorCommand.Reverse := TRUE;
	    ELSE
	        #iqUDT_LowerInfeedConveyorCommand.ManualStartStop := FALSE;
	        #iqUDT_LowerInfeedConveyorCommand.Reverse := FALSE;
	    END_IF;

	    //Lower Outfeed
	    IF #iqUDT_LiftConveyorCommand.ManualMode
	        AND #iqUDT_LowerOutfeedConveyorCommand.ManualMode
	        AND #ix_DownPosition
	        AND #ix_LiftConveyorRight
	        AND #ix_OutfeedConveyor
	    THEN
	        #iqUDT_LiftConveyorCommand.ManualStartStop := TRUE;
	        #iqUDT_LiftConveyorCommand.Reverse := FALSE;
	        #iqUDT_LowerOutfeedConveyorCommand.ManualStartStop := TRUE;
	        #iqUDT_LowerOutfeedConveyorCommand.Reverse := FALSE;

	    ELSIF #iqUDT_LiftConveyorCommand.ManualMode
	        AND #iqUDT_LowerOutfeedConveyorCommand.ManualMode
	        AND #ix_DownPosition
	        AND #ix_LiftConveyorLeft
	        AND #ix_OutfeedConveyor
	    THEN
	        #iqUDT_LiftConveyorCommand.ManualStartStop := TRUE;
	        #iqUDT_LiftConveyorCommand.Reverse := TRUE;
	        #iqUDT_LowerOutfeedConveyorCommand.ManualStartStop := TRUE;
	        #iqUDT_LowerOutfeedConveyorCommand.Reverse := TRUE;
	    ELSE
	        #iqUDT_LowerOutfeedConveyorCommand.ManualStartStop := FALSE;
	        #iqUDT_LowerOutfeedConveyorCommand.Reverse := FALSE;
	    END_IF;
	END_REGION

	REGION Upper position
	    //Upper Infeed
	    IF #iqUDT_LiftConveyorCommand.ManualMode
	        AND #iqUDT_UpperInfeedConveyorCommand.ManualMode
	        AND #ix_UpPosition
	        AND #ix_LiftConveyorLeft
	        AND #ix_InfeedConveyor
	    THEN
	        #iqUDT_LiftConveyorCommand.ManualStartStop := TRUE;
	        #iqUDT_LiftConveyorCommand.Reverse := TRUE;
	        #iqUDT_UpperInfeedConveyorCommand.ManualStartStop := TRUE;
	        #iqUDT_UpperInfeedConveyorCommand.Reverse := FALSE;

	    ELSIF #iqUDT_LiftConveyorCommand.ManualMode
	        AND #iqUDT_UpperInfeedConveyorCommand.ManualMode
	        AND #ix_UpPosition
	        AND #ix_LiftConveyorRight
	        AND #ix_InfeedConveyor
	    THEN
	        #iqUDT_LiftConveyorCommand.ManualStartStop := TRUE;
	        #iqUDT_LiftConveyorCommand.Reverse := FALSE;
	        #iqUDT_UpperInfeedConveyorCommand.ManualStartStop := TRUE;
	        #iqUDT_UpperInfeedConveyorCommand.Reverse := TRUE;
	    ELSE
	        #iqUDT_UpperInfeedConveyorCommand.ManualStartStop := FALSE;
	        #iqUDT_UpperInfeedConveyorCommand.Reverse := FALSE;
	    END_IF;

	    //Upper Outfeed
	    IF #iqUDT_LiftConveyorCommand.ManualMode
	        AND #iqUDT_UpperOutfeedConveyorCommand.ManualMode
	        AND #ix_UpPosition
	        AND #ix_LiftConveyorRight
	        AND #ix_OutfeedConveyor
	    THEN
	        #iqUDT_LiftConveyorCommand.ManualStartStop := TRUE;
	        #iqUDT_LiftConveyorCommand.Reverse := FALSE;
	        #iqUDT_UpperOutfeedConveyorCommand.ManualStartStop := TRUE;
	        #iqUDT_UpperOutfeedConveyorCommand.Reverse := TRUE;

	    ELSIF #iqUDT_LiftConveyorCommand.ManualMode
	        AND #iqUDT_UpperOutfeedConveyorCommand.ManualMode
	        AND #ix_UpPosition
	        AND #ix_LiftConveyorLeft
	        AND #ix_OutfeedConveyor
	    THEN
	        #iqUDT_LiftConveyorCommand.ManualStartStop := TRUE;
	        #iqUDT_LiftConveyorCommand.Reverse := TRUE;
	        #iqUDT_UpperOutfeedConveyorCommand.ManualStartStop := TRUE;
	        #iqUDT_UpperOutfeedConveyorCommand.Reverse := FALSE;
	    ELSE
	        #iqUDT_UpperOutfeedConveyorCommand.ManualStartStop := FALSE;
	        #iqUDT_UpperOutfeedConveyorCommand.Reverse := FALSE;
	    END_IF;
	END_REGION
END_FUNCTION_BLOCK

FUNCTION_BLOCK "FB_VfdSEWMOVI-CSpeed"
TITLE = FB_VFD_SEW_MOVI-C_Speed
{ S7_Optimized_Access := 'TRUE' }
AUTHOR : MHSE
VERSION : 3.0
// ATTRIBUTES
// AUTO_NUMBER = True
// BLOCK_NUMBER = 37
// END_ATTRIBUTES
   VAR_INPUT
      iUDT_VfdConfig { ExternalAccessible := 'False'; ExternalVisible := 'False'; ExternalWritable := 'False'} : "UDT_VfdConfiguration";   //    Configuration structure
      iUDT_VfdInputs { ExternalAccessible := 'False'; ExternalVisible := 'False'; ExternalWritable := 'False'} : "UDT_VfdSEWSpeedPI";   //    VFD inputs structure
      ix_PowerOK { ExternalAccessible := 'False'; ExternalVisible := 'False'; ExternalWritable := 'False'} : Bool;   //    True = External Power OK
      ix_SimulationModeActive { ExternalAccessible := 'False'; ExternalVisible := 'False'; ExternalWritable := 'False'} : Bool;   //    True = Simulation mode active
      ix_QuickStopDisable { ExternalAccessible := 'False'; ExternalVisible := 'False'; ExternalWritable := 'False'} : Bool := FALSE;   //    True = Quick Stop not enabled
   END_VAR

   VAR_OUTPUT
      qUDT_HMIStatus { ExternalAccessible := 'False'; ExternalVisible := 'False'; ExternalWritable := 'False'} : "UDT_VfdStatus";   //    HMI status structure
      qUDT_VfdOutputs { ExternalAccessible := 'False'; ExternalVisible := 'False'; ExternalWritable := 'False'} : "UDT_VfdSEWSpeedPO";   //    VFD outputs structure
   END_VAR

   VAR_IN_OUT
      iqUDT_ConveyorInterface : "UDT_ConveyorInterface";   //    Conveyor interface structure
      iqUDT_VfdStatistics : "UDT_VfdStatistics";   //    Statistics structure
   END_VAR

   VAR
      sUDT_HMIStatus { ExternalAccessible := 'False'; ExternalVisible := 'False'; ExternalWritable := 'False'; S7_SetPoint := 'False'} : "UDT_VfdStatus";   //    HMI status structure
      sUDT_PNDevice { ExternalAccessible := 'False'; ExternalVisible := 'False'; ExternalWritable := 'False'; S7_SetPoint := 'False'} : "UDT_PNDevice";   //    PN device info structure
      sFB_TimerOnOffDelayCheckSupply { ExternalAccessible := 'False'; ExternalVisible := 'False'; ExternalWritable := 'False'; S7_SetPoint := 'False'} : "FB_TimerOnOffDelay";   //    MHS "TimerOnOffDelay" - to delay time for VFD supply contactor
      sFB_TimerOnOffDelayMoviKit { ExternalAccessible := 'False'; ExternalVisible := 'False'; ExternalWritable := 'False'; S7_SetPoint := 'False'} : "FB_TimerOnOffDelay";   //    MHS "TimerOnOffDelay" - to delay time for MoviKit response delay error
      sFB_TimerOnOffDelayVFDRunningFeedbackError { ExternalAccessible := 'False'; ExternalVisible := 'False'; ExternalWritable := 'False'; S7_SetPoint := 'False'} : "FB_TimerOnOffDelay";   //    MHS "TimerOnOffDelay" - to delay time for VFDRunningFeedback error
      sR_TRIG_RunFWD {InstructionName := 'R_TRIG'; LibVersion := '1.0'; ExternalAccessible := 'False'; ExternalVisible := 'False'; ExternalWritable := 'False'; S7_SetPoint := 'False'} : R_TRIG;   //    Rising edge of Run forward signal
      sR_TRIG_RunRVS {InstructionName := 'R_TRIG'; LibVersion := '1.0'; ExternalAccessible := 'False'; ExternalVisible := 'False'; ExternalWritable := 'False'; S7_SetPoint := 'False'} : R_TRIG;   //    Rising edge of Run reverse
      sR_TRIG_PNSlaveNotOnline {InstructionName := 'R_TRIG'; LibVersion := '1.0'; ExternalAccessible := 'False'; ExternalVisible := 'False'; ExternalWritable := 'False'; S7_SetPoint := 'False'} : R_TRIG;   //    Rising edge for trigger Profinet slave not online statistics
      sR_TRIG_PNSlaveError {InstructionName := 'R_TRIG'; LibVersion := '1.0'; ExternalAccessible := 'False'; ExternalVisible := 'False'; ExternalWritable := 'False'; S7_SetPoint := 'False'} : R_TRIG;   //    Rising edge for trigger Profinet slave error statistics
      sR_TRIG_InternalError {InstructionName := 'R_TRIG'; LibVersion := '1.0'; ExternalAccessible := 'False'; ExternalVisible := 'False'; ExternalWritable := 'False'; S7_SetPoint := 'False'} : R_TRIG;   //    Rising edge for trigger Internal VFD Error statistics
      sR_TRIG_CommunicationErrorMovikit {InstructionName := 'R_TRIG'; LibVersion := '1.0'; ExternalAccessible := 'False'; ExternalVisible := 'False'; ExternalWritable := 'False'; S7_SetPoint := 'False'} : R_TRIG;   //    Rising edge for trigger communication error Movikit statistics
      sR_TRIG_Running {InstructionName := 'R_TRIG'; LibVersion := '1.0'; ExternalAccessible := 'False'; ExternalVisible := 'False'; ExternalWritable := 'False'; S7_SetPoint := 'False'} : R_TRIG;   //    Rising edge for starting of the running signal
      sF_TRIG_RunFwd {InstructionName := 'F_TRIG'; LibVersion := '1.0'; ExternalAccessible := 'False'; ExternalVisible := 'False'; ExternalWritable := 'False'; S7_SetPoint := 'False'} : F_TRIG;   //    Falling edge for run forward signal
      sF_TRIG_RunRvs {InstructionName := 'F_TRIG'; LibVersion := '1.0'; ExternalAccessible := 'False'; ExternalVisible := 'False'; ExternalWritable := 'False'; S7_SetPoint := 'False'} : F_TRIG;   //    Falling edge for run reverse signal
      sa_PNPortsStatus { ExternalAccessible := 'False'; ExternalVisible := 'False'; ExternalWritable := 'False'} : Array[1..8] of Bool;   // TRUE when specific port has an error
      sr_ActualSpeedSetpoint { ExternalAccessible := 'False'; ExternalVisible := 'False'; ExternalWritable := 'False'} : Real;   //    Actual speed setpoint [RPM]
      si_ActualSpeed { ExternalAccessible := 'False'; ExternalVisible := 'False'; ExternalWritable := 'False'} : Int;   //    Actual speed in [mm/s]
      sx_ConfigurationError { ExternalAccessible := 'False'; ExternalVisible := 'False'; ExternalWritable := 'False'} : Bool;   //    Commissioning: configuration error
      sx_PNDeviceHealthy { ExternalAccessible := 'False'; ExternalVisible := 'False'; ExternalWritable := 'False'} : Bool;   //    Profinet device is online and error free
      sx_MoviKitFeedback { ExternalAccessible := 'False'; ExternalVisible := 'False'; ExternalWritable := 'False'} : Bool;   //    Movikit feedback delay
      sx_HardwareAvailable { ExternalAccessible := 'False'; ExternalVisible := 'False'; ExternalWritable := 'False'} : Bool;   //    Power and communication to drive are ok
      sx_PowerOk { ExternalAccessible := 'False'; ExternalVisible := 'False'; ExternalWritable := 'False'} : Bool;   //    Communication, safety and power are available
      sx_VfdAvailable { ExternalAccessible := 'False'; ExternalVisible := 'False'; ExternalWritable := 'False'} : Bool;   //    Hardware of VFD is ok and no communication error with movikit
      sx_ErrorActive { ExternalAccessible := 'False'; ExternalVisible := 'False'; ExternalWritable := 'False'} : Bool;   //    Block has an error
      sx_EnableOperation { ExternalAccessible := 'False'; ExternalVisible := 'False'; ExternalWritable := 'False'} : Bool;   //    Enable operation signal
      sx_RunVfdForward { ExternalAccessible := 'False'; ExternalVisible := 'False'; ExternalWritable := 'False'} : Bool;   //    Start VFD forward
      sx_RunVfdReverse { ExternalAccessible := 'False'; ExternalVisible := 'False'; ExternalWritable := 'False'} : Bool;   //    Start VFD backward
      sx_SpeedSetpointReached { ExternalAccessible := 'False'; ExternalVisible := 'False'; ExternalWritable := 'False'} : Bool;   //    Motor is running at requested speed
      sx_VfdStopping { ExternalAccessible := 'False'; ExternalVisible := 'False'; ExternalWritable := 'False'} : Bool;   //    VFD Stopping
      sx_MovikitHandshakeIn { ExternalAccessible := 'False'; ExternalVisible := 'False'; ExternalWritable := 'False'} : Bool;   //    Handshake to movikit
   END_VAR

   VAR CONSTANT
      ci_NumberOfProfinetPorts : Int := 2;   // Number of Profinet ports in device
   END_VAR


BEGIN
	(*
	----------------------------------------------------------------------------------------

	Version history:
	Date        | Version   | Author        | Remark
	----------------------------------------------------------------------------------------
	24/05/2019  | 0.1       | P. Majka      | First release MHS TIA 15.1
	24/07/2019  | 0.2       | K. Pokorski   | Autofind device is Profinet structure (Region 2)
	30/07/2019  | 0.3       | M. Kurc       | Add MoviKit error
	30/07/2019  | 2.0       | P. Majka      | Moved to project with library 2.0
	16/08/2019  | 2.1       | T.v.Beukering | Updated complete block
	03/10/2019  | 2.2       | F.Baten       | Applied FC_GetDevicePN, added running statistics, changed speed window from UInt to Int, added actual speed in conveyor interface.
	11/10/2019  | 2.3       | M. Kurc       | Added VFD stop signal when occurs both run request (FWD, RVS), added logic for QuickSTOP, added interclok FDW/RVS
	20/11/2019  | 2.10      | S. Nikodem    | Configuration error
	20/11/2019  | 3.0       | P.Majka       | 3.0 MHS library release TIA 15.1
	03/12/2019  | 3.1       | S. Nikodem    | Change of direction
	20/12/2019  | 3.2       | S. Deulkar    | Used configureation error bit to report to conveyor block
	06/02/2020  | 3.3       | S. Nikodem    | Configuration error - Simulation mode bypass PNDeviceFound
	01/03/2020  | 3.4       | F.Baten       | Changed "UDT_VFD_Status" to be without positioning status
	04/03/2020  | 3.5       | F.Baten       | Output speed scaling based on measured speed at fixed output value, removal of gearratio and wheelendperrimeter
	01/05/2020  | 3.7       | F.Baten       | Reverted 3.6 modification measured speed
	14/09/2020  | 3.8       | S.Nikodem     | VFDRunningFeedback error
	03/11/2020  | 3.9       | K.Pokorski    | Profinet ports diagnostics added
	21/02/2023  | 4.0       | F.Baten       | 4.0 Release TIA 17.5
	*)

	REGION 1 - Get Device Profinet information

	    "FC_GetDevicePN"(is_PNDeviceName := #iUDT_VfdConfig.VFDPNDeviceName,
	                     ix_SimulationModeActive := #ix_SimulationModeActive,
	                     iqUDT_PND := #sUDT_PNDevice);


	    "FC_GetPNPortStatus"(ii_NumberOfPorts := #ci_NumberOfProfinetPorts,
	                         iUDT_DevicePNInfo := #sUDT_PNDevice,
	                         qa_PortFault => #sa_PNPortsStatus);

	END_REGION

	REGION 2 - Reset errors

	    IF #iqUDT_ConveyorInterface.InternalErrorReset                           // Reset errors when reset signal is given
	    THEN
	        #sUDT_HMIStatus.CommunicationErrorMovikit := FALSE;
	        #sUDT_HMIStatus.PNSlaveNotonline := FALSE;
	        #sUDT_HMIStatus.PNSlaveError := FALSE;
	        #sUDT_HMIStatus.InternalError := FALSE;
	        #sUDT_HMIStatus.VFDRunningFeedbackError := FALSE;
	        #sUDT_HMIStatus.PNSlaveWarning := FALSE;

	    END_IF;

	END_REGION

	REGION 3 - Hardware checks
	    // Hardware will only be available after the delay, so the device has time for the initialisation
	    #sFB_TimerOnOffDelayCheckSupply(iudi_OnDelayTime := 2000,
	                                    ix_SignalToDelay := #ix_PowerOK);

	    #sx_PowerOk := #sFB_TimerOnOffDelayCheckSupply.qx_DelayedSignal;

	    // Check if PN device is online
	    IF NOT "DB_ProfinetDiagnostic".ProfinetNetworks[#sUDT_PNDevice.PNNetworknumber].DeviceStatus[#sUDT_PNDevice.PNDeviceNumber].DeviceState.Exist
	        AND NOT #ix_SimulationModeActive
	        AND #sx_PowerOk
	    THEN
	        #sUDT_HMIStatus.PNSlaveNotonline := TRUE;
	    END_IF;


	    // Check if PN ports are healthy
	    IF #sa_PNPortsStatus[1] XOR #sa_PNPortsStatus[2] THEN
	        #sUDT_HMIStatus.PNSlaveWarning := TRUE;
	    END_IF;

	    // Check if PN device has an error
	    IF "DB_ProfinetDiagnostic".ProfinetNetworks[#sUDT_PNDevice.PNNetworknumber].DeviceStatus[#sUDT_PNDevice.PNDeviceNumber].DeviceState.Error
	        AND NOT #ix_SimulationModeActive
	        AND #sx_PowerOk
	        AND NOT #sUDT_HMIStatus.PNSlaveWarning
	    THEN
	        #sUDT_HMIStatus.PNSlaveError := TRUE;
	    END_IF;

	    // Set bit when PN device is healthy (online and no error)
	    #sx_PNDeviceHealthy := NOT #sUDT_HMIStatus.PNSlaveNotonline
	    AND NOT #sUDT_HMIStatus.PNSlaveError
	    AND #sUDT_PNDevice.PNDeviceFound
	    AND #sx_PowerOk;

	    // Set hardware available bit when all conditions are met
	    #sx_HardwareAvailable := (#iUDT_VfdInputs.Status_Word_1.STO_Inactive
	    AND #sx_PowerOk
	    AND #sx_PNDeviceHealthy)
	    OR #ix_SimulationModeActive;

	    // Check MoviKit communication (heartbeat)
	    #sx_MoviKitFeedback := ((#sx_MovikitHandshakeIn
	    AND NOT #iUDT_VfdInputs.Status_Word_1.MovikitHandshakeOut)
	    OR (NOT #sx_MovikitHandshakeIn
	    AND #iUDT_VfdInputs.Status_Word_1.MovikitHandshakeOut));

	    #sFB_TimerOnOffDelayMoviKit(iudi_OnDelayTime := 1000,
	                                ix_SignalToDelay := NOT #sx_MoviKitFeedback);

	    // Set error when MoviKit communication is not available
	    IF #sFB_TimerOnOffDelayMoviKit.qx_DelayedSignal AND #sx_HardwareAvailable
	    THEN

	        #sUDT_HMIStatus.CommunicationErrorMovikit := TRUE;

	    END_IF;

	    // Invert output when input is equal
	    #sx_MovikitHandshakeIn := NOT #iUDT_VfdInputs.Status_Word_1.MovikitHandshakeOut;

	    // VFD is ready for operation if hardware ok and no communication error with Movikit
	    #sx_VfdAvailable := #sx_HardwareAvailable AND NOT #sUDT_HMIStatus.CommunicationErrorMovikit;

	END_REGION

	REGION 4 - Check errors and warnings
	    // Check if the VFD has an error
	    #sUDT_HMIStatus.InternalError := #iUDT_VfdInputs.Status_Word_1.Error;

	    // Check if the VFD has a warning
	    #sUDT_HMIStatus.InternalWarning := #iUDT_VfdInputs.Status_Word_1.Warning;

	    // Copy error/warning code to status DB when error/warning active
	    IF NOT #iUDT_VfdInputs.Status_Word_1.Error
	        AND NOT #iUDT_VfdInputs.Status_Word_1.Warning
	    THEN
	        #sUDT_HMIStatus.ErrorCode := 0;
	        #sUDT_HMIStatus.SubErrorCode := 0;
	    ELSE
	        #sUDT_HMIStatus.ErrorCode := #iUDT_VfdInputs.StatusErrorNo.%B1;
	        #sUDT_HMIStatus.SubErrorCode := #iUDT_VfdInputs.StatusErrorNo.%B0;
	    END_IF;

	END_REGION

	REGION 5 - Check if configuration is ok for commissioning purposes
	    // Set configuration error when one or all VFD configuration parameters aren't set
	    IF #iUDT_VfdConfig.WheelEndPerimeter > 0.0
	        AND #iUDT_VfdConfig.GearRatio > 0.0
	        AND #iUDT_VfdConfig.ReferenceRPM > 0.0
	        AND #iUDT_VfdConfig.VFDStartupTime > 0.0
	        AND (#sUDT_PNDevice.PNDeviceFound
	        OR #ix_SimulationModeActive)
	    THEN
	        #sx_ConfigurationError := FALSE;
	    ELSE
	        #sx_ConfigurationError := TRUE;

	    END_IF;

	END_REGION

	REGION 6 - Handle speed
	    // Calculate speed in mm/s
	    #si_ActualSpeed := REAL_TO_INT(((#iUDT_VfdInputs.ActualSpeed / #iUDT_VfdConfig.GearRatio) * #iUDT_VfdConfig.WheelEndPerimeter) / 60.0);

	    // Reversal direction speed
	    IF #iUDT_VfdConfig.DirectionReversal
	    THEN
	        #si_ActualSpeed := #si_ActualSpeed * -1;

	    END_IF;

	    // Actual speed setpoint
	    #sr_ActualSpeedSetpoint := ((DINT_TO_REAL(INT_TO_DINT(#iqUDT_ConveyorInterface.SpeedSetpoint) * 60) / #iUDT_VfdConfig.WheelEndPerimeter) * #iUDT_VfdConfig.GearRatio);

	    // Check maximum output
	    IF
	        #sr_ActualSpeedSetpoint > #iUDT_VfdConfig.ReferenceRPM
	    THEN
	        #sr_ActualSpeedSetpoint := #iUDT_VfdConfig.ReferenceRPM;
	    END_IF;


	    //Check if speed setpoint is reached
	    #sx_SpeedSetpointReached := (ABS(#si_ActualSpeed) >= (#iqUDT_ConveyorInterface.SpeedSetpoint - #iUDT_VfdConfig.SpeedSetpointWindow))
	    AND (ABS(#si_ActualSpeed) <= (#iqUDT_ConveyorInterface.SpeedSetpoint + #iUDT_VfdConfig.SpeedSetpointWindow));


	END_REGION

